   1:  PR[91,2] = PR[90,2] + 18.690;
   1:  PR[91,3] = PR[90,3] + 110.566;
   1:L PR[91] R[100]mm/sec CNT100;
   1:  PR[91,1] = PR[90,1] + -21.590;
   1:  PR[91,2] = PR[90,2] + 15.011;
   1:  PR[91,3] = PR[90,3] + 110.605;
   1:L PR[91] R[100]mm/sec CNT100;
   1:  PR[91,1] = PR[90,1] + -26.072;
   1:  PR[91,2] = PR[90,2] + 11.127;
   1:  PR[91,3] = PR[90,3] + 110.640;
   1:L PR[91] R[100]mm/sec CNT100;
   1:  PR[91,1] = PR[90,1] + -28.046;
   1:  PR[91,2] = PR[90,2] + 8.636;
   1:  PR[91,3] = PR[90,3] + 110.670;
   1:L PR[91] R[100]mm/sec CNT100;
   1:  PR[91,1] = PR[90,1] + -29.203;
   1:  PR[91,2] = PR[90,2] + 7.162;
   1:  PR[91,3] = PR[90,3] + 110.686;
   1:L PR[91] R[100]mm/sec CNT100;
   1:  PR[91] = PR[90];
   1:  PR[91,1] = PR[90,1] + -28.899;
   1:  PR[91,2] = PR[90,2] + 3.219;
   1:  PR[91,3] = PR[90,3] + 111.995;
   1:L PR[91] R[100]mm/sec CNT100;
   1:  PR[91,1] = PR[90,1] + -29.295;
   1:  PR[91,2] = PR[90,2] + 0.620;
   1:  PR[91,3] = PR[90,3] + 110.717;
   1:L PR[91] R[100]mm/sec CNT100;
   1:  PR[91,1] = PR[90,1] + -29.499;
   1:  PR[91,2] = PR[90,2] + -0.729;
   1:  PR[91,3] = PR[90,3] + 110.731;
   1:L PR[91] R[100]mm/sec CNT100;
   1:  PR[91,1] = PR[90,1] + -28.898;
   1:  PR[91,2] = PR[90,2] + -4.678;
   1:  PR[91,3] = PR[90,3] + 110.738;
   1:L PR[91] R[100]mm/sec CNT100;
   1:  PR[91,1] = PR[90,1] + -27.056;
   1:  PR[91,2] = PR[90,2] + -8.680;
   1:  PR[91,3] = PR[90,3] + 110.758;
   1:L PR[91] R[100]mm/sec CNT100;
   1:  PR[91,1] = PR[90,1] + -23.900;
   1:  PR[91,2] = PR[90,2] + -12.680;
   1:  PR[91,3] = PR[90,3] + 110.780;
   1:L PR[91] R[100]mm/sec CNT100;
   1:  PR[91,1] = PR[90,1] + -21.408;
   1:  PR[91,2] = PR[90,2] + -14.850;
   1:  PR[91,3] = PR[90,3] + 110.806;
   1:L PR[91] R[100]mm/sec CNT100;
   1:  PR[91,1] = PR[90,1] + -19.393;
   1:  PR[91,2] = PR[90,2] + -16.589;
   1:  PR[91,3] = PR[90,3] + 110.823;
   1:L PR[91] R[100]mm/sec CNT100;
   1:  PR[91,1] = PR[90,1] + -13.560;
   1:  PR[91,2] = PR[90,2] + -20.296;
   1:  PR[91,3] = PR[90,3] + 110.836;
   1:L PR[91] R[100]mm/sec CNT100;
   1:  PR[91,1] = PR[90,1] + -6.447;
   1:  PR[91,2] = PR[90,2] + -23.694;
   1:  PR[91,3] = PR[90,3] + 110.871;
   1:L PR[91] R[100]mm/sec CNT100;
   1:  PR[91,1] = PR[90,1] + -0.885;
   1:  PR[91,2] = PR[90,2] + -25.699;
   1:  PR[91,3] = PR[90,3] + 110.911;
   1:L PR[91] R[100]mm/sec CNT100;
   1:  PR[91,1] = PR[90,1] + 0.617;
   1:  PR[91,2] = PR[90,2] + -26.345;
   1:  PR[91,3] = PR[90,3] + 110.941;
   1:L PR[91] R[100]mm/sec CNT100;
   1:  PR[91,1] = PR[90,1] + 2.242;
   1:  PR[91,2] = PR[90,2] + -26.979;
   1:  PR[91,3] = PR[90,3] + 110.950;
   1:L PR[91] R[100]mm/sec CNT100;
   1:  PR[91,1] = PR[90,1] + 5.927;
   1:  PR[91,2] = PR[90,2] + -28.163;
   1:  PR[91,3] = PR[90,3] + 110.959;
   1:L PR[91] R[100]mm/sec CNT100;
   1:  PR[91,1] = PR[90,1] + 10.541;
   1:  PR[91,2] = PR[90,2] + -29.357;
   1:  PR[91,3] = PR[90,3] + 110.978;
   1:L PR[91] R[100]mm/sec CNT100;
   1:  PR[91,1] = PR[90,1] + 13.547;
   1:  PR[91,2] = PR[90,2] + -30.335;
   1:  PR[91,3] = PR[90,3] + 111.002;
   1:L PR[91] R[100]mm/sec CNT100;
   1:  PR[91,1] = PR[90,1] + 22.631;
   1:  PR[91,2] = PR[90,2] + -32.054;
   1:  PR[91,3] = PR[90,3] + 111.018;
   1:L PR[91] R[100]mm/sec CNT100;
   1:  PR[91,1] = PR[90,1] + 31.896;
   1:  PR[91,2] = PR[90,2] + -32.675;
   1:  PR[91,3] = PR[90,3] + 111.065;
   1:L PR[91] R[100]mm/sec CNT100;
   1:  PR[91,1] = PR[90,1] + 35.449;
   1:  PR[91,2] = PR[90,2] + -32.699;
   1:  PR[91,3] = PR[90,3] + 111.112;
   1:L PR[91] R[100]mm/sec CNT100;
   1:  PR[91,1] = PR[90,1] + 37.094;
   1:  PR[91,2] = PR[90,2] + -32.535;
   1:  PR[91,3] = PR[90,3] + 111.130;
   1:L PR[91] R[100]mm/sec CNT100;
   1:  PR[91,1] = PR[90,1] + 42.048;
   1:  PR[91,2] = PR[90,2] + -31.700;
   1:  PR[91,3] = PR[90,3] + 111.139;
   1:L PR[91] R[100]mm/sec CNT100;
   1:  PR[91,1] = PR[90,1] + 42.311;
   1:  PR[91,2] = PR[90,2] + -31.628;
   1:  PR[91,3] = PR[90,3] + 111.164;
   1:L PR[91] R[100]mm/sec CNT100;
   1:  PR[91,1] = PR[90,1] + 43.722;
   1:  PR[91,2] = PR[90,2] + -31.123;
   1:  PR[91,3] = PR[90,3] + 111.166;
   1:L PR[91] R[100]mm/sec CNT100;
   1:  PR[91,1] = PR[90,1] + 48.274;
   1:  PR[91,2] = PR[90,2] + -29.546;
   1:  PR[91,3] = PR[90,3] + 111.173;
   1:L PR[91] R[100]mm/sec CNT100;
   1:  PR[91,1] = PR[90,1] + 53.963;
   1:  PR[91,2] = PR[90,2] + -26.403;
   1:  PR[91,3] = PR[90,3] + 111.198;
   1:L PR[91] R[100]mm/sec CNT100;
   1:  PR[91,1] = PR[90,1] + 56.746;
   1:  PR[91,2] = PR[90,2] + -24.164;
   1:  PR[91,3] = PR[90,3] + 111.231;
   1:L PR[91] R[100]mm/sec CNT100;
   1:  PR[91,1] = PR[90,1] + 58.567;
   1:  PR[91,2] = PR[90,2] + -22.765;
   1:  PR[91,3] = PR[90,3] + 111.249;
   1:L PR[91] R[100]mm/sec CNT100;
   1:  PR[91,1] = PR[90,1] + 59.454;
   1:  PR[91,2] = PR[90,2] + -21.955;
   1:  PR[91,3] = PR[90,3] + 111.261;
   1:L PR[91] R[100]mm/sec CNT100;
   1:  PR[91,1] = PR[90,1] + 61.281;
   1:  PR[91,2] = PR[90,2] + -19.912;
   1:  PR[91,3] = PR[90,3] + 111.267;
   1:L PR[91] R[100]mm/sec CNT100;
   1:  PR[91,1] = PR[90,1] + 63.248;
   1:  PR[91,2] = PR[90,2] + -17.593;
   1:  PR[91,3] = PR[90,3] + 111.281;
   1:L PR[91] R[100]mm/sec CNT100;
   1:  PR[91,1] = PR[90,1] + 65.653;
   1:  PR[91,2] = PR[90,2] + -13.713;
   1:  PR[91,3] = PR[90,3] + 111.296;
   1:L PR[91] R[100]mm/sec CNT100;
   1:  PR[91,1] = PR[90,1] + 67.493;
   1:  PR[91,2] = PR[90,2] + -9.389;
   1:  PR[91,3] = PR[90,3] + 111.319;
   1:L PR[91] R[100]mm/sec CNT100;
   1:  PR[91,1] = PR[90,1] + 68.495;
   1:  PR[91,2] = PR[90,2] + -5.359;
   1:  PR[91,3] = PR[90,3] + 111.343;
   1:L PR[91] R[100]mm/sec CNT100;
   1:  PR[91,1] = PR[90,1] + 68.842;
   1:  PR[91,2] = PR[90,2] + -1.092;
   1:  PR[91,3] = PR[90,3] + 111.364;
   1:L PR[91] R[100]mm/sec CNT100;
   1:  PR[91,1] = PR[90,1] + 68.902;
   1:  PR[91,2] = PR[90,2] + -0.670;
   1:  PR[91,3] = PR[90,3] + 111.386;
   1:L PR[91] R[100]mm/sec CNT100;
   1:  PR[91,1] = PR[90,1] + 68.564;
   1:  PR[91,2] = PR[90,2] + 3.453;
   1:  PR[91,3] = PR[90,3] + 111.388;
   1:L PR[91] R[100]mm/sec CNT100;
   1:  PR[91,1] = PR[90,1] + 68.509;
   1:  PR[91,2] = PR[90,2] + 3.843;
   1:  PR[91,3] = PR[90,3] + 111.409;
   1:L PR[91] R[100]mm/sec CNT100;
   1:  PR[91,1] = PR[90,1] + 67.493;
   1:  PR[91,2] = PR[90,2] + 7.930;
   1:  PR[91,3] = PR[90,3] + 111.411;
   1:L PR[91] R[100]mm/sec CNT100;
   1:  PR[91,1] = PR[90,1] + 65.654;
   1:  PR[91,2] = PR[90,2] + 12.253;
   1:  PR[91,3] = PR[90,3] + 111.432;
   1:L PR[91] R[100]mm/sec CNT100;
   1:  PR[91,1] = PR[90,1] + 63.250;
   1:  PR[91,2] = PR[90,2] + 16.132;
   1:  PR[91,3] = PR[90,3] + 111.456;
   1:L PR[91] R[100]mm/sec CNT100;
   1:  PR[91,1] = PR[90,1] + 61.281;
   1:  PR[91,2] = PR[90,2] + 18.453;
   1:  PR[91,3] = PR[90,3] + 111.479;
   1:L PR[91] R[100]mm/sec CNT100;
   1:  PR[91,1] = PR[90,1] + 59.452;
   1:  PR[91,2] = PR[90,2] + 20.498;
   1:  PR[91,3] = PR[90,3] + 111.495;
   1:L PR[91] R[100]mm/sec CNT100;
   1:  PR[91,1] = PR[90,1] + 58.565;
   1:  PR[91,2] = PR[90,2] + 21.308;
   1:  PR[91,3] = PR[90,3] + 111.509;
   1:L PR[91] R[100]mm/sec CNT100;
   1:  PR[91,1] = PR[90,1] + 56.747;
   1:  PR[91,2] = PR[90,2] + 22.706;
   1:  PR[91,3] = PR[90,3] + 111.515;
   1:L PR[91] R[100]mm/sec CNT100;
   1:  PR[91,1] = PR[90,1] + 53.961;
   1:  PR[91,2] = PR[90,2] + 24.947;
   1:  PR[91,3] = PR[90,3] + 111.526;
   1:L PR[91] R[100]mm/sec CNT100;
   1:  PR[91,1] = PR[90,1] + 48.276;
   1:  PR[91,2] = PR[90,2] + 28.086;
   1:  PR[91,3] = PR[90,3] + 111.544;
   1:L PR[91] R[100]mm/sec CNT100;
   1:  PR[91,1] = PR[90,1] + 43.722;
   1:  PR[91,2] = PR[90,2] + 29.664;
   1:  PR[91,3] = PR[90,3] + 111.577;
   1:L PR[91] R[100]mm/sec CNT100;
   1:  PR[91,1] = PR[90,1] + 42.315;
   1:  PR[91,2] = PR[90,2] + 30.169;
   1:  PR[91,3] = PR[90,3] + 111.602;
   1:L PR[91] R[100]mm/sec CNT100;
   1:  PR[91,1] = PR[90,1] + 42.054;
   1:  PR[91,2] = PR[90,2] + 30.240;
   1:  PR[91,3] = PR[90,3] + 111.609;
   1:L PR[91] R[100]mm/sec CNT100;
   1:  PR[91,1] = PR[90,1] + 37.093;
   1:  PR[91,2] = PR[90,2] + 31.077;
   1:  PR[91,3] = PR[90,3] + 111.611;
   1:L PR[91] R[100]mm/sec CNT100;
   1:  PR[91,1] = PR[90,1] + 35.447;
   1:  PR[91,2] = PR[90,2] + 31.240;
   1:  PR[91,3] = PR[90,3] + 111.636;
   1:L PR[91] R[100]mm/sec CNT100;
   1:  PR[91,1] = PR[90,1] + 31.881;
   1:  PR[91,2] = PR[90,2] + 31.216;
   1:  PR[91,3] = PR[90,3] + 111.645;
   1:L PR[91] R[100]mm/sec CNT100;
   1:  PR[91,1] = PR[90,1] + 22.655;
   1:  PR[91,2] = PR[90,2] + 30.598;
   1:  PR[91,3] = PR[90,3] + 111.663;
   1:L PR[91] R[100]mm/sec CNT100;
   1:  PR[91,1] = PR[90,1] + 13.553;
   1:  PR[91,2] = PR[90,2] + 28.878;
   1:  PR[91,3] = PR[90,3] + 111.710;
   1:L PR[91] R[100]mm/sec CNT100;
   1:  PR[91,1] = PR[90,1] + 10.541;
   1:  PR[91,2] = PR[90,2] + 27.899;
   1:  PR[91,3] = PR[90,3] + 111.757;
   1:L PR[91] R[100]mm/sec CNT100;
   1:  PR[91,1] = PR[90,1] + 5.928;
   1:  PR[91,2] = PR[90,2] + 26.705;
   1:  PR[91,3] = PR[90,3] + 111.773;
   1:L PR[91] R[100]mm/sec CNT100;
   1:  PR[91,1] = PR[90,1] + 2.242;
   1:  PR[91,2] = PR[90,2] + 25.520;
   1:  PR[91,3] = PR[90,3] + 111.797;
   1:L PR[91] R[100]mm/sec CNT100;
   1:  PR[91,1] = PR[90,1] + 0.617;
   1:  PR[91,2] = PR[90,2] + 24.886;
   1:  PR[91,3] = PR[90,3] + 111.817;
   1:L PR[91] R[100]mm/sec CNT100;
   1:  PR[91,1] = PR[90,1] + -0.885;
   1:  PR[91,2] = PR[90,2] + 24.240;
   1:  PR[91,3] = PR[90,3] + 111.826;
   1:L PR[91] R[100]mm/sec CNT100;
   1:  PR[91,1] = PR[90,1] + -6.447;
   1:  PR[91,2] = PR[90,2] + 22.236;
   1:  PR[91,3] = PR[90,3] + 111.834;
   1:L PR[91] R[100]mm/sec CNT100;
   1:  PR[91,1] = PR[90,1] + -13.560;
   1:  PR[91,2] = PR[90,2] + 18.838;
   1:  PR[91,3] = PR[90,3] + 111.864;
   1:L PR[91] R[100]mm/sec CNT100;
   1:  PR[91,1] = PR[90,1] + -19.393;
   1:  PR[91,2] = PR[90,2] + 15.130;
   1:  PR[91,3] = PR[90,3] + 111.904;
   1:L PR[91] R[100]mm/sec CNT100;
   1:  PR[91,1] = PR[90,1] + -21.408;
   1:  PR[91,2] = PR[90,2] + 13.392;
   1:  PR[91,3] = PR[90,3] + 111.939;
   1:L PR[91] R[100]mm/sec CNT100;
   1:  PR[91,1] = PR[90,1] + -23.900;
   1:  PR[91,2] = PR[90,2] + 11.222;
   1:  PR[91,3] = PR[90,3] + 111.952;
   1:L PR[91] R[100]mm/sec CNT100;
   1:  PR[91,1] = PR[90,1] + -27.057;
   1:  PR[91,2] = PR[90,2] + 7.221;
   1:  PR[91,3] = PR[90,3] + 111.969;
   1:L PR[91] R[100]mm/sec CNT100;
   1:  PR[91] = PR[90];
   1:  PR[91,1] = PR[90,1] + -26.764;
   1:  PR[91,2] = PR[90,2] + 3.250;
   1:  PR[91,3] = PR[90,3] + 113.295;
   1:L PR[91] R[100]mm/sec CNT100;
   1:  PR[91,1] = PR[90,1] + -27.119;
   1:  PR[91,2] = PR[90,2] + 0.925;
   1:  PR[91,3] = PR[90,3] + 112.018;
   1:L PR[91] R[100]mm/sec CNT100;
   1:  PR[91,1] = PR[90,1] + -27.369;
   1:  PR[91,2] = PR[90,2] + -0.729;
   1:  PR[91,3] = PR[90,3] + 112.030;
   1:L PR[91] R[100]mm/sec CNT100;
   1:  PR[91,1] = PR[90,1] + -26.763;
   1:  PR[91,2] = PR[90,2] + -4.710;
   1:  PR[91,3] = PR[90,3] + 112.038;
   1:L PR[91] R[100]mm/sec CNT100;
   1:  PR[91,1] = PR[90,1] + -24.908;
   1:  PR[91,2] = PR[90,2] + -8.742;
   1:  PR[91,3] = PR[90,3] + 112.059;
   1:L PR[91] R[100]mm/sec CNT100;
   1:  PR[91,1] = PR[90,1] + -21.730;
   1:  PR[91,2] = PR[90,2] + -12.772;
   1:  PR[91,3] = PR[90,3] + 112.082;
   1:L PR[91] R[100]mm/sec CNT100;
   1:  PR[91,1] = PR[90,1] + -18.889;
   1:  PR[91,2] = PR[90,2] + -15.247;
   1:  PR[91,3] = PR[90,3] + 112.108;
   1:L PR[91] R[100]mm/sec CNT100;
   1:  PR[91,1] = PR[90,1] + -17.193;
   1:  PR[91,2] = PR[90,2] + -16.710;
   1:  PR[91,3] = PR[90,3] + 112.127;
   1:L PR[91] R[100]mm/sec CNT100;
   1:  PR[91,1] = PR[90,1] + -11.322;
   1:  PR[91,2] = PR[90,2] + -20.444;
   1:  PR[91,3] = PR[90,3] + 112.139;
   1:L PR[91] R[100]mm/sec CNT100;
   1:  PR[91,1] = PR[90,1] + -4.162;
   1:  PR[91,2] = PR[90,2] + -23.867;
   1:  PR[91,3] = PR[90,3] + 112.174;
   1:L PR[91] R[100]mm/sec CNT100;
   1:  PR[91,1] = PR[90,1] + -1.534;
   1:  PR[91,2] = PR[90,2] + -24.815;
   1:  PR[91,3] = PR[90,3] + 112.215;
   1:L PR[91] R[100]mm/sec CNT100;
   1:  PR[91,1] = PR[90,1] + 1.504;
   1:  PR[91,2] = PR[90,2] + -26.121;
   1:  PR[91,3] = PR[90,3] + 112.229;
   1:L PR[91] R[100]mm/sec CNT100;
   1:  PR[91,1] = PR[90,1] + 4.908;
   1:  PR[91,2] = PR[90,2] + -27.449;
   1:  PR[91,3] = PR[90,3] + 112.246;
   1:L PR[91] R[100]mm/sec CNT100;
   1:  PR[91,1] = PR[90,1] + 6.995;
   1:  PR[91,2] = PR[90,2] + -28.120;
   1:  PR[91,3] = PR[90,3] + 112.265;
   1:L PR[91] R[100]mm/sec CNT100;
   1:  PR[91,1] = PR[90,1] + 9.670;
   1:  PR[91,2] = PR[90,2] + -28.812;
   1:  PR[91,3] = PR[90,3] + 112.276;
   1:L PR[91] R[100]mm/sec CNT100;
   1:  PR[91,1] = PR[90,1] + 15.006;
   1:  PR[91,2] = PR[90,2] + -30.547;
   1:  PR[91,3] = PR[90,3] + 112.290;
   1:L PR[91] R[100]mm/sec CNT100;
   1:  PR[91,1] = PR[90,1] + 23.781;
   1:  PR[91,2] = PR[90,2] + -32.216;
   1:  PR[91,3] = PR[90,3] + 112.319;
   1:L PR[91] R[100]mm/sec CNT100;
   1:  PR[91,1] = PR[90,1] + 24.941;
   1:  PR[91,2] = PR[90,2] + -32.331;
   1:  PR[91,3] = PR[90,3] + 112.365;
   1:L PR[91] R[100]mm/sec CNT100;
   1:  PR[91,1] = PR[90,1] + 31.610;
   1:  PR[91,2] = PR[90,2] + -32.779;
   1:  PR[91,3] = PR[90,3] + 112.371;
   1:L PR[91] R[100]mm/sec CNT100;
   1:  PR[91,1] = PR[90,1] + 36.265;
   1:  PR[91,2] = PR[90,2] + -32.811;
   1:  PR[91,3] = PR[90,3] + 112.405;
   1:L PR[91] R[100]mm/sec CNT100;
   1:  PR[91,1] = PR[90,1] + 36.806;
   1:  PR[91,2] = PR[90,2] + -32.757;
   1:  PR[91,3] = PR[90,3] + 112.429;
   1:L PR[91] R[100]mm/sec CNT100;
   1:  PR[91,1] = PR[90,1] + 42.786;
   1:  PR[91,2] = PR[90,2] + -31.760;
   1:  PR[91,3] = PR[90,3] + 112.431;
   1:L PR[91] R[100]mm/sec CNT100;
   1:  PR[91,1] = PR[90,1] + 48.989;
   1:  PR[91,2] = PR[90,2] + -29.610;
   1:  PR[91,3] = PR[90,3] + 112.462;
   1:L PR[91] R[100]mm/sec CNT100;
   1:  PR[91,1] = PR[90,1] + 50.842;
   1:  PR[91,2] = PR[90,2] + -28.581;
   1:  PR[91,3] = PR[90,3] + 112.496;
   1:L PR[91] R[100]mm/sec CNT100;
   1:  PR[91,1] = PR[90,1] + 54.708;
   1:  PR[91,2] = PR[90,2] + -26.471;
   1:  PR[91,3] = PR[90,3] + 112.507;
   1:L PR[91] R[100]mm/sec CNT100;
   1:  PR[91,1] = PR[90,1] + 54.975;
   1:  PR[91,2] = PR[90,2] + -26.285;
   1:  PR[91,3] = PR[90,3] + 112.529;
   1:L PR[91] R[100]mm/sec CNT100;
   1:  PR[91,1] = PR[90,1] + 58.574;
   1:  PR[91,2] = PR[90,2] + -23.518;
   1:  PR[91,3] = PR[90,3] + 112.531;
   1:L PR[91] R[100]mm/sec CNT100;
   1:  PR[91,1] = PR[90,1] + 60.968;
   1:  PR[91,2] = PR[90,2] + -21.332;
   1:  PR[91,3] = PR[90,3] + 112.554;
   1:L PR[91] R[100]mm/sec CNT100;
   1:  PR[91,1] = PR[90,1] + 64.170;
   1:  PR[91,2] = PR[90,2] + -17.527;
   1:  PR[91,3] = PR[90,3] + 112.571;
   1:L PR[91] R[100]mm/sec CNT100;
   1:  PR[91,1] = PR[90,1] + 66.488;
   1:  PR[91,2] = PR[90,2] + -13.787;
   1:  PR[91,3] = PR[90,3] + 112.596;
   1:L PR[91] R[100]mm/sec CNT100;
   1:  PR[91,1] = PR[90,1] + 68.141;
   1:  PR[91,2] = PR[90,2] + -9.880;
   1:  PR[91,3] = PR[90,3] + 112.619;
   1:L PR[91] R[100]mm/sec CNT100;
   1:  PR[91,1] = PR[90,1] + 68.387;
   1:  PR[91,2] = PR[90,2] + -9.331;
   1:  PR[91,3] = PR[90,3] + 112.641;
   1:L PR[91] R[100]mm/sec CNT100;
   1:  PR[91,1] = PR[90,1] + 69.347;
   1:  PR[91,2] = PR[90,2] + -5.468;
   1:  PR[91,3] = PR[90,3] + 112.644;
   1:L PR[91] R[100]mm/sec CNT100;
   1:  PR[91,1] = PR[90,1] + 69.682;
   1:  PR[91,2] = PR[90,2] + -1.352;
   1:  PR[91,3] = PR[90,3] + 112.664;
   1:L PR[91] R[100]mm/sec CNT100;
   1:  PR[91,1] = PR[90,1] + 69.778;
   1:  PR[91,2] = PR[90,2] + -0.670;
   1:  PR[91,3] = PR[90,3] + 112.685;
   1:L PR[91] R[100]mm/sec CNT100;
   1:  PR[91,1] = PR[90,1] + 69.454;
   1:  PR[91,2] = PR[90,2] + 3.301;
   1:  PR[91,3] = PR[90,3] + 112.689;
   1:L PR[91] R[100]mm/sec CNT100;
   1:  PR[91,1] = PR[90,1] + 69.361;
   1:  PR[91,2] = PR[90,2] + 3.952;
   1:  PR[91,3] = PR[90,3] + 112.709;
   1:L PR[91] R[100]mm/sec CNT100;
   1:  PR[91,1] = PR[90,1] + 68.383;
   1:  PR[91,2] = PR[90,2] + 7.888;
   1:  PR[91,3] = PR[90,3] + 112.712;
   1:L PR[91] R[100]mm/sec CNT100;
   1:  PR[91,1] = PR[90,1] + 66.490;
   1:  PR[91,2] = PR[90,2] + 12.325;
   1:  PR[91,3] = PR[90,3] + 112.733;
   1:L PR[91] R[100]mm/sec CNT100;
   1:  PR[91,1] = PR[90,1] + 64.172;
   1:  PR[91,2] = PR[90,2] + 16.066;
   1:  PR[91,3] = PR[90,3] + 112.758;
   1:L PR[91] R[100]mm/sec CNT100;
   1:  PR[91,1] = PR[90,1] + 60.970;
   1:  PR[91,2] = PR[90,2] + 19.870;
   1:  PR[91,3] = PR[90,3] + 112.780;
   1:L PR[91] R[100]mm/sec CNT100;
   1:  PR[91,1] = PR[90,1] + 58.573;
   1:  PR[91,2] = PR[90,2] + 22.060;
   1:  PR[91,3] = PR[90,3] + 112.806;
   1:L PR[91] R[100]mm/sec CNT100;
   1:  PR[91,1] = PR[90,1] + 54.968;
   1:  PR[91,2] = PR[90,2] + 24.831;
   1:  PR[91,3] = PR[90,3] + 112.822;
   1:L PR[91] R[100]mm/sec CNT100;
   1:  PR[91,1] = PR[90,1] + 54.704;
   1:  PR[91,2] = PR[90,2] + 25.015;
   1:  PR[91,3] = PR[90,3] + 112.846;
   1:L PR[91] R[100]mm/sec CNT100;
   1:  PR[91,1] = PR[90,1] + 50.840;
   1:  PR[91,2] = PR[90,2] + 27.123;
   1:  PR[91,3] = PR[90,3] + 112.847;
   1:L PR[91] R[100]mm/sec CNT100;
   1:  PR[91,1] = PR[90,1] + 48.987;
   1:  PR[91,2] = PR[90,2] + 28.153;
   1:  PR[91,3] = PR[90,3] + 112.870;
   1:L PR[91] R[100]mm/sec CNT100;
   1:  PR[91,1] = PR[90,1] + 42.790;
   1:  PR[91,2] = PR[90,2] + 30.300;
   1:  PR[91,3] = PR[90,3] + 112.881;
   1:L PR[91] R[100]mm/sec CNT100;
   1:  PR[91,1] = PR[90,1] + 36.810;
   1:  PR[91,2] = PR[90,2] + 31.298;
   1:  PR[91,3] = PR[90,3] + 112.914;
   1:L PR[91] R[100]mm/sec CNT100;
   1:  PR[91,1] = PR[90,1] + 36.270;
   1:  PR[91,2] = PR[90,2] + 31.351;
   1:  PR[91,3] = PR[90,3] + 112.945;
   1:L PR[91] R[100]mm/sec CNT100;
   1:  PR[91,1] = PR[90,1] + 31.596;
   1:  PR[91,2] = PR[90,2] + 31.320;
   1:  PR[91,3] = PR[90,3] + 112.948;
   1:L PR[91] R[100]mm/sec CNT100;
   1:  PR[91,1] = PR[90,1] + 24.966;
   1:  PR[91,2] = PR[90,2] + 30.875;
   1:  PR[91,3] = PR[90,3] + 112.972;
   1:L PR[91] R[100]mm/sec CNT100;
   1:  PR[91,1] = PR[90,1] + 24.303;
   1:  PR[91,2] = PR[90,2] + 30.818;
   1:  PR[91,3] = PR[90,3] + 113.006;
   1:L PR[91] R[100]mm/sec CNT100;
   1:  PR[91,1] = PR[90,1] + 23.813;
   1:  PR[91,2] = PR[90,2] + 30.762;
   1:  PR[91,3] = PR[90,3] + 113.009;
   1:L PR[91] R[100]mm/sec CNT100;
   1:  PR[91,1] = PR[90,1] + 15.015;
   1:  PR[91,2] = PR[90,2] + 29.091;
   1:  PR[91,3] = PR[90,3] + 113.012;
   1:L PR[91] R[100]mm/sec CNT100;
   1:  PR[91,1] = PR[90,1] + 9.670;
   1:  PR[91,2] = PR[90,2] + 27.353;
   1:  PR[91,3] = PR[90,3] + 113.058;
   1:L PR[91] R[100]mm/sec CNT100;
   1:  PR[91,1] = PR[90,1] + 6.996;
   1:  PR[91,2] = PR[90,2] + 26.661;
   1:  PR[91,3] = PR[90,3] + 113.086;
   1:L PR[91] R[100]mm/sec CNT100;
   1:  PR[91,1] = PR[90,1] + 4.909;
   1:  PR[91,2] = PR[90,2] + 25.990;
   1:  PR[91,3] = PR[90,3] + 113.101;
   1:L PR[91] R[100]mm/sec CNT100;
   1:  PR[91,1] = PR[90,1] + 1.504;
   1:  PR[91,2] = PR[90,2] + 24.663;
   1:  PR[91,3] = PR[90,3] + 113.112;
   1:L PR[91] R[100]mm/sec CNT100;
   1:  PR[91,1] = PR[90,1] + -1.534;
   1:  PR[91,2] = PR[90,2] + 23.356;
   1:  PR[91,3] = PR[90,3] + 113.131;
   1:L PR[91] R[100]mm/sec CNT100;
   1:  PR[91,1] = PR[90,1] + -4.162;
   1:  PR[91,2] = PR[90,2] + 22.408;
   1:  PR[91,3] = PR[90,3] + 113.147;
   1:L PR[91] R[100]mm/sec CNT100;
   1:  PR[91,1] = PR[90,1] + -11.322;
   1:  PR[91,2] = PR[90,2] + 18.985;
   1:  PR[91,3] = PR[90,3] + 113.162;
   1:L PR[91] R[100]mm/sec CNT100;
   1:  PR[91,1] = PR[90,1] + -17.193;
   1:  PR[91,2] = PR[90,2] + 15.251;
   1:  PR[91,3] = PR[90,3] + 113.202;
   1:L PR[91] R[100]mm/sec CNT100;
   1:  PR[91,1] = PR[90,1] + -18.889;
   1:  PR[91,2] = PR[90,2] + 13.788;
   1:  PR[91,3] = PR[90,3] + 113.238;
   1:L PR[91] R[100]mm/sec CNT100;
   1:  PR[91,1] = PR[90,1] + -21.730;
   1:  PR[91,2] = PR[90,2] + 11.313;
   1:  PR[91,3] = PR[90,3] + 113.249;
   1:L PR[91] R[100]mm/sec CNT100;
   1:  PR[91,1] = PR[90,1] + -24.908;
   1:  PR[91,2] = PR[90,2] + 7.283;
   1:  PR[91,3] = PR[90,3] + 113.269;
   1:L PR[91] R[100]mm/sec CNT100;
   1:  PR[91] = PR[90];
   1:  PR[91,1] = PR[90,1] + -24.629;
   1:  PR[91,2] = PR[90,2] + 3.281;
   1:  PR[91,3] = PR[90,3] + 114.595;
   1:L PR[91] R[100]mm/sec CNT100;
   1:  PR[91,1] = PR[90,1] + -24.942;
   1:  PR[91,2] = PR[90,2] + 1.230;
   1:  PR[91,3] = PR[90,3] + 113.318;
   1:L PR[91] R[100]mm/sec CNT100;
   1:  PR[91,1] = PR[90,1] + -25.238;
   1:  PR[91,2] = PR[90,2] + -0.729;
   1:  PR[91,3] = PR[90,3] + 113.329;
   1:L PR[91] R[100]mm/sec CNT100;
   1:  PR[91,1] = PR[90,1] + -24.628;
   1:  PR[91,2] = PR[90,2] + -4.741;
   1:  PR[91,3] = PR[90,3] + 113.339;
   1:L PR[91] R[100]mm/sec CNT100;
   1:  PR[91,1] = PR[90,1] + -22.760;
   1:  PR[91,2] = PR[90,2] + -8.804;
   1:  PR[91,3] = PR[90,3] + 113.360;
   1:L PR[91] R[100]mm/sec CNT100;
   1:  PR[91,1] = PR[90,1] + -19.561;
   1:  PR[91,2] = PR[90,2] + -12.863;
   1:  PR[91,3] = PR[90,3] + 113.383;
   1:L PR[91] R[100]mm/sec CNT100;
   1:  PR[91,1] = PR[90,1] + -16.370;
   1:  PR[91,2] = PR[90,2] + -15.643;
   1:  PR[91,3] = PR[90,3] + 113.410;
   1:L PR[91] R[100]mm/sec CNT100;
   1:  PR[91,1] = PR[90,1] + -14.994;
   1:  PR[91,2] = PR[90,2] + -16.830;
   1:  PR[91,3] = PR[90,3] + 113.432;
   1:L PR[91] R[100]mm/sec CNT100;
   1:  PR[91,1] = PR[90,1] + -9.084;
   1:  PR[91,2] = PR[90,2] + -20.592;
   1:  PR[91,3] = PR[90,3] + 113.441;
   1:L PR[91] R[100]mm/sec CNT100;
   1:  PR[91,1] = PR[90,1] + -1.996;
   1:  PR[91,2] = PR[90,2] + -23.983;
   1:  PR[91,3] = PR[90,3] + 113.477;
   1:L PR[91] R[100]mm/sec CNT100;
   1:  PR[91,1] = PR[90,1] + -1.787;
   1:  PR[91,2] = PR[90,2] + -24.100;
   1:  PR[91,3] = PR[90,3] + 113.518;
   1:L PR[91] R[100]mm/sec CNT100;
   1:  PR[91,1] = PR[90,1] + 2.391;
   1:  PR[91,2] = PR[90,2] + -25.898;
   1:  PR[91,3] = PR[90,3] + 113.519;
   1:L PR[91] R[100]mm/sec CNT100;
   1:  PR[91,1] = PR[90,1] + 7.574;
   1:  PR[91,2] = PR[90,2] + -27.919;
   1:  PR[91,3] = PR[90,3] + 113.542;
   1:L PR[91] R[100]mm/sec CNT100;
   1:  PR[91,1] = PR[90,1] + 8.064;
   1:  PR[91,2] = PR[90,2] + -28.076;
   1:  PR[91,3] = PR[90,3] + 113.571;
   1:L PR[91] R[100]mm/sec CNT100;
   1:  PR[91,1] = PR[90,1] + 8.798;
   1:  PR[91,2] = PR[90,2] + -28.266;
   1:  PR[91,3] = PR[90,3] + 113.574;
   1:L PR[91] R[100]mm/sec CNT100;
   1:  PR[91,1] = PR[90,1] + 16.462;
   1:  PR[91,2] = PR[90,2] + -30.759;
   1:  PR[91,3] = PR[90,3] + 113.578;
   1:L PR[91] R[100]mm/sec CNT100;
   1:  PR[91,1] = PR[90,1] + 21.916;
   1:  PR[91,2] = PR[90,2] + -31.791;
   1:  PR[91,3] = PR[90,3] + 113.619;
   1:L PR[91] R[100]mm/sec CNT100;
   1:  PR[91,1] = PR[90,1] + 24.452;
   1:  PR[91,2] = PR[90,2] + -32.298;
   1:  PR[91,3] = PR[90,3] + 113.648;
   1:L PR[91] R[100]mm/sec CNT100;
   1:  PR[91,1] = PR[90,1] + 26.635;
   1:  PR[91,2] = PR[90,2] + -32.539;
   1:  PR[91,3] = PR[90,3] + 113.661;
   1:L PR[91] R[100]mm/sec CNT100;
   1:  PR[91,1] = PR[90,1] + 28.358;
   1:  PR[91,2] = PR[90,2] + -32.684;
   1:  PR[91,3] = PR[90,3] + 113.673;
   1:L PR[91] R[100]mm/sec CNT100;
   1:  PR[91,1] = PR[90,1] + 31.324;
   1:  PR[91,2] = PR[90,2] + -32.883;
   1:  PR[91,3] = PR[90,3] + 113.682;
   1:L PR[91] R[100]mm/sec CNT100;
   1:  PR[91,1] = PR[90,1] + 36.319;
   1:  PR[91,2] = PR[90,2] + -32.920;
   1:  PR[91,3] = PR[90,3] + 113.697;
   1:L PR[91] R[100]mm/sec CNT100;
   1:  PR[91,1] = PR[90,1] + 36.948;
   1:  PR[91,2] = PR[90,2] + -32.915;
   1:  PR[91,3] = PR[90,3] + 113.723;
   1:L PR[91] R[100]mm/sec CNT100;
   1:  PR[91,1] = PR[90,1] + 43.475;
   1:  PR[91,2] = PR[90,2] + -31.834;
   1:  PR[91,3] = PR[90,3] + 113.726;
   1:L PR[91] R[100]mm/sec CNT100;
   1:  PR[91,1] = PR[90,1] + 49.712;
   1:  PR[91,2] = PR[90,2] + -29.672;
   1:  PR[91,3] = PR[90,3] + 113.760;
   1:L PR[91] R[100]mm/sec CNT100;
   1:  PR[91,1] = PR[90,1] + 54.252;
   1:  PR[91,2] = PR[90,2] + -27.185;
   1:  PR[91,3] = PR[90,3] + 113.794;
   1:L PR[91] R[100]mm/sec CNT100;
   1:  PR[91,1] = PR[90,1] + 55.099;
   1:  PR[91,2] = PR[90,2] + -26.774;
   1:  PR[91,3] = PR[90,3] + 113.821;
   1:L PR[91] R[100]mm/sec CNT100;
   1:  PR[91,1] = PR[90,1] + 57.508;
   1:  PR[91,2] = PR[90,2] + -25.095;
   1:  PR[91,3] = PR[90,3] + 113.826;
   1:L PR[91] R[100]mm/sec CNT100;
   1:  PR[91,1] = PR[90,1] + 58.585;
   1:  PR[91,2] = PR[90,2] + -24.267;
   1:  PR[91,3] = PR[90,3] + 113.841;
   1:L PR[91] R[100]mm/sec CNT100;
   1:  PR[91,1] = PR[90,1] + 61.855;
   1:  PR[91,2] = PR[90,2] + -21.320;
   1:  PR[91,3] = PR[90,3] + 113.848;
   1:L PR[91] R[100]mm/sec CNT100;
   1:  PR[91,1] = PR[90,1] + 65.093;
   1:  PR[91,2] = PR[90,2] + -17.458;
   1:  PR[91,3] = PR[90,3] + 113.871;
   1:L PR[91] R[100]mm/sec CNT100;
   1:  PR[91,1] = PR[90,1] + 67.323;
   1:  PR[91,2] = PR[90,2] + -13.860;
   1:  PR[91,3] = PR[90,3] + 113.897;
   1:L PR[91] R[100]mm/sec CNT100;
   1:  PR[91,1] = PR[90,1] + 68.916;
   1:  PR[91,2] = PR[90,2] + -10.097;
   1:  PR[91,3] = PR[90,3] + 113.918;
   1:L PR[91] R[100]mm/sec CNT100;
   1:  PR[91,1] = PR[90,1] + 69.276;
   1:  PR[91,2] = PR[90,2] + -9.290;
   1:  PR[91,3] = PR[90,3] + 113.940;
   1:L PR[91] R[100]mm/sec CNT100;
   1:  PR[91,1] = PR[90,1] + 70.199;
   1:  PR[91,2] = PR[90,2] + -5.578;
   1:  PR[91,3] = PR[90,3] + 113.944;
   1:L PR[91] R[100]mm/sec CNT100;
   1:  PR[91,1] = PR[90,1] + 70.522;
   1:  PR[91,2] = PR[90,2] + -1.612;
   1:  PR[91,3] = PR[90,3] + 113.964;
   1:L PR[91] R[100]mm/sec CNT100;
   1:  PR[91,1] = PR[90,1] + 70.655;
   1:  PR[91,2] = PR[90,2] + -0.670;
   1:  PR[91,3] = PR[90,3] + 113.984;
   1:L PR[91] R[100]mm/sec CNT100;
   1:  PR[91,1] = PR[90,1] + 70.343;
   1:  PR[91,2] = PR[90,2] + 3.149;
   1:  PR[91,3] = PR[90,3] + 113.989;
   1:L PR[91] R[100]mm/sec CNT100;
   1:  PR[91,1] = PR[90,1] + 70.213;
   1:  PR[91,2] = PR[90,2] + 4.062;
   1:  PR[91,3] = PR[90,3] + 114.009;
   1:L PR[91] R[100]mm/sec CNT100;
   1:  PR[91,1] = PR[90,1] + 69.272;
   1:  PR[91,2] = PR[90,2] + 7.850;
   1:  PR[91,3] = PR[90,3] + 114.014;
   1:L PR[91] R[100]mm/sec CNT100;
   1:  PR[91,1] = PR[90,1] + 67.626;
   1:  PR[91,2] = PR[90,2] + 11.730;
   1:  PR[91,3] = PR[90,3] + 114.034;
   1:L PR[91] R[100]mm/sec CNT100;
   1:  PR[91,1] = PR[90,1] + 67.334;
   1:  PR[91,2] = PR[90,2] + 12.383;
   1:  PR[91,3] = PR[90,3] + 114.056;
   1:L PR[91] R[100]mm/sec CNT100;
   1:  PR[91,1] = PR[90,1] + 65.095;
   1:  PR[91,2] = PR[90,2] + 15.997;
   1:  PR[91,3] = PR[90,3] + 114.059;
   1:L PR[91] R[100]mm/sec CNT100;
   1:  PR[91,1] = PR[90,1] + 61.858;
   1:  PR[91,2] = PR[90,2] + 19.859;
   1:  PR[91,3] = PR[90,3] + 114.081;
   1:L PR[91] R[100]mm/sec CNT100;
   1:  PR[91,1] = PR[90,1] + 58.587;
   1:  PR[91,2] = PR[90,2] + 22.807;
   1:  PR[91,3] = PR[90,3] + 114.107;
   1:L PR[91] R[100]mm/sec CNT100;
   1:  PR[91,1] = PR[90,1] + 57.509;
   1:  PR[91,2] = PR[90,2] + 23.636;
   1:  PR[91,3] = PR[90,3] + 114.130;
   1:L PR[91] R[100]mm/sec CNT100;
   1:  PR[91,1] = PR[90,1] + 55.067;
   1:  PR[91,2] = PR[90,2] + 25.337;
   1:  PR[91,3] = PR[90,3] + 114.137;
   1:L PR[91] R[100]mm/sec CNT100;
   1:  PR[91,1] = PR[90,1] + 51.454;
   1:  PR[91,2] = PR[90,2] + 27.253;
   1:  PR[91,3] = PR[90,3] + 114.153;
   1:L PR[91] R[100]mm/sec CNT100;
   1:  PR[91,1] = PR[90,1] + 49.704;
   1:  PR[91,2] = PR[90,2] + 28.217;
   1:  PR[91,3] = PR[90,3] + 114.174;
   1:L PR[91] R[100]mm/sec CNT100;
   1:  PR[91,1] = PR[90,1] + 43.475;
   1:  PR[91,2] = PR[90,2] + 30.375;
   1:  PR[91,3] = PR[90,3] + 114.184;
   1:L PR[91] R[100]mm/sec CNT100;
   1:  PR[91,1] = PR[90,1] + 36.954;
   1:  PR[91,2] = PR[90,2] + 31.456;
   1:  PR[91,3] = PR[90,3] + 114.218;
   1:L PR[91] R[100]mm/sec CNT100;
   1:  PR[91,1] = PR[90,1] + 36.297;
   1:  PR[91,2] = PR[90,2] + 31.460;
   1:  PR[91,3] = PR[90,3] + 114.252;
   1:L PR[91] R[100]mm/sec CNT100;
   1:  PR[91,1] = PR[90,1] + 31.313;
   1:  PR[91,2] = PR[90,2] + 31.424;
   1:  PR[91,3] = PR[90,3] + 114.255;
   1:L PR[91] R[100]mm/sec CNT100;
   1:  PR[91,1] = PR[90,1] + 28.387;
   1:  PR[91,2] = PR[90,2] + 31.228;
   1:  PR[91,3] = PR[90,3] + 114.281;
   1:L PR[91] R[100]mm/sec CNT100;
   1:  PR[91,1] = PR[90,1] + 26.210;
   1:  PR[91,2] = PR[90,2] + 31.040;
   1:  PR[91,3] = PR[90,3] + 114.296;
   1:L PR[91] R[100]mm/sec CNT100;
   1:  PR[91,1] = PR[90,1] + 24.471;
   1:  PR[91,2] = PR[90,2] + 30.841;
   1:  PR[91,3] = PR[90,3] + 114.308;
   1:L PR[91] R[100]mm/sec CNT100;
   1:  PR[91,1] = PR[90,1] + 21.916;
   1:  PR[91,2] = PR[90,2] + 30.332;
   1:  PR[91,3] = PR[90,3] + 114.317;
   1:L PR[91] R[100]mm/sec CNT100;
   1:  PR[91,1] = PR[90,1] + 16.475;
   1:  PR[91,2] = PR[90,2] + 29.304;
   1:  PR[91,3] = PR[90,3] + 114.330;
   1:L PR[91] R[100]mm/sec CNT100;
   1:  PR[91,1] = PR[90,1] + 8.798;
   1:  PR[91,2] = PR[90,2] + 26.807;
   1:  PR[91,3] = PR[90,3] + 114.359;
   1:L PR[91] R[100]mm/sec CNT100;
   1:  PR[91,1] = PR[90,1] + 8.064;
   1:  PR[91,2] = PR[90,2] + 26.617;
   1:  PR[91,3] = PR[90,3] + 114.400;
   1:L PR[91] R[100]mm/sec CNT100;
   1:  PR[91,1] = PR[90,1] + 7.575;
   1:  PR[91,2] = PR[90,2] + 26.460;
   1:  PR[91,3] = PR[90,3] + 114.404;
   1:L PR[91] R[100]mm/sec CNT100;
   1:  PR[91,1] = PR[90,1] + 2.390;
   1:  PR[91,2] = PR[90,2] + 24.439;
   1:  PR[91,3] = PR[90,3] + 114.407;
   1:L PR[91] R[100]mm/sec CNT100;
   1:  PR[91,1] = PR[90,1] + -1.787;
   1:  PR[91,2] = PR[90,2] + 22.642;
   1:  PR[91,3] = PR[90,3] + 114.436;
   1:L PR[91] R[100]mm/sec CNT100;
   1:  PR[91,1] = PR[90,1] + -1.996;
   1:  PR[91,2] = PR[90,2] + 22.524;
   1:  PR[91,3] = PR[90,3] + 114.459;
   1:L PR[91] R[100]mm/sec CNT100;
   1:  PR[91,1] = PR[90,1] + -9.084;
   1:  PR[91,2] = PR[90,2] + 19.133;
   1:  PR[91,3] = PR[90,3] + 114.460;
   1:L PR[91] R[100]mm/sec CNT100;
   1:  PR[91,1] = PR[90,1] + -14.994;
   1:  PR[91,2] = PR[90,2] + 15.371;
   1:  PR[91,3] = PR[90,3] + 114.501;
   1:L PR[91] R[100]mm/sec CNT100;
   1:  PR[91,1] = PR[90,1] + -16.370;
   1:  PR[91,2] = PR[90,2] + 14.184;
   1:  PR[91,3] = PR[90,3] + 114.537;
   1:L PR[91] R[100]mm/sec CNT100;
   1:  PR[91,1] = PR[90,1] + -19.561;
   1:  PR[91,2] = PR[90,2] + 11.405;
   1:  PR[91,3] = PR[90,3] + 114.546;
   1:L PR[91] R[100]mm/sec CNT100;
   1:  PR[91,1] = PR[90,1] + -22.760;
   1:  PR[91,2] = PR[90,2] + 7.345;
   1:  PR[91,3] = PR[90,3] + 114.568;
   1:L PR[91] R[100]mm/sec CNT100;
   1:  PR[91] = PR[90];
   1:  PR[91,1] = PR[90,1] + -22.494;
   1:  PR[91,2] = PR[90,2] + 3.312;
   1:  PR[91,3] = PR[90,3] + 115.895;
   1:L PR[91] R[100]mm/sec CNT100;
   1:  PR[91,1] = PR[90,1] + -22.765;
   1:  PR[91,2] = PR[90,2] + 1.535;
   1:  PR[91,3] = PR[90,3] + 114.618;
   1:L PR[91] R[100]mm/sec CNT100;
   1:  PR[91,1] = PR[90,1] + -23.108;
   1:  PR[91,2] = PR[90,2] + -0.729;
   1:  PR[91,3] = PR[90,3] + 114.628;
   1:L PR[91] R[100]mm/sec CNT100;
   1:  PR[91,1] = PR[90,1] + -22.494;
   1:  PR[91,2] = PR[90,2] + -4.772;
   1:  PR[91,3] = PR[90,3] + 114.640;
   1:L PR[91] R[100]mm/sec CNT100;
   1:  PR[91,1] = PR[90,1] + -20.612;
   1:  PR[91,2] = PR[90,2] + -8.866;
   1:  PR[91,3] = PR[90,3] + 114.661;
   1:L PR[91] R[100]mm/sec CNT100;
   1:  PR[91,1] = PR[90,1] + -17.392;
   1:  PR[91,2] = PR[90,2] + -12.955;
   1:  PR[91,3] = PR[90,3] + 114.684;
   1:L PR[91] R[100]mm/sec CNT100;
   1:  PR[91,1] = PR[90,1] + -13.851;
   1:  PR[91,2] = PR[90,2] + -16.039;
   1:  PR[91,3] = PR[90,3] + 114.712;
   1:L PR[91] R[100]mm/sec CNT100;
   1:  PR[91,1] = PR[90,1] + -12.794;
   1:  PR[91,2] = PR[90,2] + -16.950;
   1:  PR[91,3] = PR[90,3] + 114.736;
   1:L PR[91] R[100]mm/sec CNT100;
   1:  PR[91,1] = PR[90,1] + -6.846;
   1:  PR[91,2] = PR[90,2] + -20.739;
   1:  PR[91,3] = PR[90,3] + 114.743;
   1:L PR[91] R[100]mm/sec CNT100;
   1:  PR[91,1] = PR[90,1] + -2.644;
   1:  PR[91,2] = PR[90,2] + -22.750;
   1:  PR[91,3] = PR[90,3] + 114.780;
   1:L PR[91] R[100]mm/sec CNT100;
   1:  PR[91,1] = PR[90,1] + 0.246;
   1:  PR[91,2] = PR[90,2] + -24.370;
   1:  PR[91,3] = PR[90,3] + 114.804;
   1:L PR[91] R[100]mm/sec CNT100;
   1:  PR[91,1] = PR[90,1] + 3.277;
   1:  PR[91,2] = PR[90,2] + -25.674;
   1:  PR[91,3] = PR[90,3] + 114.821;
   1:L PR[91] R[100]mm/sec CNT100;
   1:  PR[91,1] = PR[90,1] + 8.168;
   1:  PR[91,2] = PR[90,2] + -27.581;
   1:  PR[91,3] = PR[90,3] + 114.839;
   1:L PR[91] R[100]mm/sec CNT100;
   1:  PR[91,1] = PR[90,1] + 9.532;
   1:  PR[91,2] = PR[90,2] + -28.245;
   1:  PR[91,3] = PR[90,3] + 114.866;
   1:L PR[91] R[100]mm/sec CNT100;
   1:  PR[91,1] = PR[90,1] + 17.919;
   1:  PR[91,2] = PR[90,2] + -30.971;
   1:  PR[91,3] = PR[90,3] + 114.874;
   1:L PR[91] R[100]mm/sec CNT100;
   1:  PR[91,1] = PR[90,1] + 20.778;
   1:  PR[91,2] = PR[90,2] + -31.512;
   1:  PR[91,3] = PR[90,3] + 114.920;
   1:L PR[91] R[100]mm/sec CNT100;
   1:  PR[91,1] = PR[90,1] + 25.106;
   1:  PR[91,2] = PR[90,2] + -32.377;
   1:  PR[91,3] = PR[90,3] + 114.935;
   1:L PR[91] R[100]mm/sec CNT100;
   1:  PR[91,1] = PR[90,1] + 28.106;
   1:  PR[91,2] = PR[90,2] + -32.720;
   1:  PR[91,3] = PR[90,3] + 114.958;
   1:L PR[91] R[100]mm/sec CNT100;
   1:  PR[91,1] = PR[90,1] + 31.231;
   1:  PR[91,2] = PR[90,2] + -32.991;
   1:  PR[91,3] = PR[90,3] + 114.974;
   1:L PR[91] R[100]mm/sec CNT100;
   1:  PR[91,1] = PR[90,1] + 35.510;
   1:  PR[91,2] = PR[90,2] + -33.023;
   1:  PR[91,3] = PR[90,3] + 114.990;
   1:L PR[91] R[100]mm/sec CNT100;
   1:  PR[91,1] = PR[90,1] + 37.610;
   1:  PR[91,2] = PR[90,2] + -33.001;
   1:  PR[91,3] = PR[90,3] + 115.012;
   1:L PR[91] R[100]mm/sec CNT100;
   1:  PR[91,1] = PR[90,1] + 41.288;
   1:  PR[91,2] = PR[90,2] + -32.398;
   1:  PR[91,3] = PR[90,3] + 115.023;
   1:L PR[91] R[100]mm/sec CNT100;
   1:  PR[91,1] = PR[90,1] + 44.160;
   1:  PR[91,2] = PR[90,2] + -31.910;
   1:  PR[91,3] = PR[90,3] + 115.043;
   1:L PR[91] R[100]mm/sec CNT100;
   1:  PR[91,1] = PR[90,1] + 50.466;
   1:  PR[91,2] = PR[90,2] + -29.725;
   1:  PR[91,3] = PR[90,3] + 115.058;
   1:L PR[91] R[100]mm/sec CNT100;
   1:  PR[91,1] = PR[90,1] + 53.807;
   1:  PR[91,2] = PR[90,2] + -27.903;
   1:  PR[91,3] = PR[90,3] + 115.092;
   1:L PR[91] R[100]mm/sec CNT100;
   1:  PR[91,1] = PR[90,1] + 55.452;
   1:  PR[91,2] = PR[90,2] + -27.103;
   1:  PR[91,3] = PR[90,3] + 115.112;
   1:L PR[91] R[100]mm/sec CNT100;
   1:  PR[91,1] = PR[90,1] + 59.146;
   1:  PR[91,2] = PR[90,2] + -24.541;
   1:  PR[91,3] = PR[90,3] + 115.122;
   1:L PR[91] R[100]mm/sec CNT100;
   1:  PR[91,1] = PR[90,1] + 62.684;
   1:  PR[91,2] = PR[90,2] + -21.367;
   1:  PR[91,3] = PR[90,3] + 115.145;
   1:L PR[91] R[100]mm/sec CNT100;
   1:  PR[91,1] = PR[90,1] + 66.017;
   1:  PR[91,2] = PR[90,2] + -17.388;
   1:  PR[91,3] = PR[90,3] + 115.170;
   1:L PR[91] R[100]mm/sec CNT100;
   1:  PR[91,1] = PR[90,1] + 68.159;
   1:  PR[91,2] = PR[90,2] + -13.932;
   1:  PR[91,3] = PR[90,3] + 115.197;
   1:L PR[91] R[100]mm/sec CNT100;
   1:  PR[91,1] = PR[90,1] + 69.690;
   1:  PR[91,2] = PR[90,2] + -10.313;
   1:  PR[91,3] = PR[90,3] + 115.218;
   1:L PR[91] R[100]mm/sec CNT100;
   1:  PR[91,1] = PR[90,1] + 70.166;
   1:  PR[91,2] = PR[90,2] + -9.249;
   1:  PR[91,3] = PR[90,3] + 115.239;
   1:L PR[91] R[100]mm/sec CNT100;
   1:  PR[91,1] = PR[90,1] + 71.051;
   1:  PR[91,2] = PR[90,2] + -5.687;
   1:  PR[91,3] = PR[90,3] + 115.245;
   1:L PR[91] R[100]mm/sec CNT100;
   1:  PR[91,1] = PR[90,1] + 71.362;
   1:  PR[91,2] = PR[90,2] + -1.872;
   1:  PR[91,3] = PR[90,3] + 115.264;
   1:L PR[91] R[100]mm/sec CNT100;
   1:  PR[91,1] = PR[90,1] + 71.532;
   1:  PR[91,2] = PR[90,2] + -0.670;
   1:  PR[91,3] = PR[90,3] + 115.284;
   1:L PR[91] R[100]mm/sec CNT100;
   1:  PR[91,1] = PR[90,1] + 71.232;
   1:  PR[91,2] = PR[90,2] + 2.997;
   1:  PR[91,3] = PR[90,3] + 115.290;
   1:L PR[91] R[100]mm/sec CNT100;
   1:  PR[91,1] = PR[90,1] + 71.066;
   1:  PR[91,2] = PR[90,2] + 4.171;
   1:  PR[91,3] = PR[90,3] + 115.309;
   1:L PR[91] R[100]mm/sec CNT100;
   1:  PR[91,1] = PR[90,1] + 70.161;
   1:  PR[91,2] = PR[90,2] + 7.809;
   1:  PR[91,3] = PR[90,3] + 115.315;
   1:L PR[91] R[100]mm/sec CNT100;
   1:  PR[91,1] = PR[90,1] + 68.579;
   1:  PR[91,2] = PR[90,2] + 11.539;
   1:  PR[91,3] = PR[90,3] + 115.335;
   1:L PR[91] R[100]mm/sec CNT100;
   1:  PR[91,1] = PR[90,1] + 68.170;
   1:  PR[91,2] = PR[90,2] + 12.455;
   1:  PR[91,3] = PR[90,3] + 115.356;
   1:L PR[91] R[100]mm/sec CNT100;
   1:  PR[91,1] = PR[90,1] + 66.019;
   1:  PR[91,2] = PR[90,2] + 15.927;
   1:  PR[91,3] = PR[90,3] + 115.361;
   1:L PR[91] R[100]mm/sec CNT100;
   1:  PR[91,1] = PR[90,1] + 62.686;
   1:  PR[91,2] = PR[90,2] + 19.907;
   1:  PR[91,3] = PR[90,3] + 115.382;
   1:L PR[91] R[100]mm/sec CNT100;
   1:  PR[91,1] = PR[90,1] + 59.148;
   1:  PR[91,2] = PR[90,2] + 23.080;
   1:  PR[91,3] = PR[90,3] + 115.409;
   1:L PR[91] R[100]mm/sec CNT100;
   1:  PR[91,1] = PR[90,1] + 55.422;
   1:  PR[91,2] = PR[90,2] + 25.665;
   1:  PR[91,3] = PR[90,3] + 115.434;
   1:L PR[91] R[100]mm/sec CNT100;
   1:  PR[91,1] = PR[90,1] + 51.801;
   1:  PR[91,2] = PR[90,2] + 27.585;
   1:  PR[91,3] = PR[90,3] + 115.458;
   1:L PR[91] R[100]mm/sec CNT100;
   1:  PR[91,1] = PR[90,1] + 50.484;
   1:  PR[91,2] = PR[90,2] + 28.261;
   1:  PR[91,3] = PR[90,3] + 115.479;
   1:L PR[91] R[100]mm/sec CNT100;
   1:  PR[91,1] = PR[90,1] + 44.159;
   1:  PR[91,2] = PR[90,2] + 30.451;
   1:  PR[91,3] = PR[90,3] + 115.487;
   1:L PR[91] R[100]mm/sec CNT100;
   1:  PR[91,1] = PR[90,1] + 37.610;
   1:  PR[91,2] = PR[90,2] + 31.542;
   1:  PR[91,3] = PR[90,3] + 115.522;
   1:L PR[91] R[100]mm/sec CNT100;
   1:  PR[91,1] = PR[90,1] + 35.516;
   1:  PR[91,2] = PR[90,2] + 31.564;
   1:  PR[91,3] = PR[90,3] + 115.556;
   1:L PR[91] R[100]mm/sec CNT100;
   1:  PR[91,1] = PR[90,1] + 31.229;
   1:  PR[91,2] = PR[90,2] + 31.532;
   1:  PR[91,3] = PR[90,3] + 115.567;
   1:L PR[91] R[100]mm/sec CNT100;
   1:  PR[91,1] = PR[90,1] + 28.118;
   1:  PR[91,2] = PR[90,2] + 31.263;
   1:  PR[91,3] = PR[90,3] + 115.590;
   1:L PR[91] R[100]mm/sec CNT100;
   1:  PR[91,1] = PR[90,1] + 25.120;
   1:  PR[91,2] = PR[90,2] + 30.920;
   1:  PR[91,3] = PR[90,3] + 115.606;
   1:L PR[91] R[100]mm/sec CNT100;
   1:  PR[91,1] = PR[90,1] + 20.777;
   1:  PR[91,2] = PR[90,2] + 30.053;
   1:  PR[91,3] = PR[90,3] + 115.621;
   1:L PR[91] R[100]mm/sec CNT100;
   1:  PR[91,1] = PR[90,1] + 17.936;
   1:  PR[91,2] = PR[90,2] + 29.517;
   1:  PR[91,3] = PR[90,3] + 115.645;
   1:L PR[91] R[100]mm/sec CNT100;
   1:  PR[91,1] = PR[90,1] + 9.535;
   1:  PR[91,2] = PR[90,2] + 26.787;
   1:  PR[91,3] = PR[90,3] + 115.660;
   1:L PR[91] R[100]mm/sec CNT100;
   1:  PR[91,1] = PR[90,1] + 8.168;
   1:  PR[91,2] = PR[90,2] + 26.122;
   1:  PR[91,3] = PR[90,3] + 115.706;
   1:L PR[91] R[100]mm/sec CNT100;
   1:  PR[91,1] = PR[90,1] + 3.277;
   1:  PR[91,2] = PR[90,2] + 24.215;
   1:  PR[91,3] = PR[90,3] + 115.713;
   1:L PR[91] R[100]mm/sec CNT100;
   1:  PR[91,1] = PR[90,1] + 0.247;
   1:  PR[91,2] = PR[90,2] + 22.911;
   1:  PR[91,3] = PR[90,3] + 115.741;
   1:L PR[91] R[100]mm/sec CNT100;
   1:  PR[91,1] = PR[90,1] + -2.644;
   1:  PR[91,2] = PR[90,2] + 21.291;
   1:  PR[91,3] = PR[90,3] + 115.758;
   1:L PR[91] R[100]mm/sec CNT100;
   1:  PR[91,1] = PR[90,1] + -6.846;
   1:  PR[91,2] = PR[90,2] + 19.280;
   1:  PR[91,3] = PR[90,3] + 115.775;
   1:L PR[91] R[100]mm/sec CNT100;
   1:  PR[91,1] = PR[90,1] + -12.794;
   1:  PR[91,2] = PR[90,2] + 15.492;
   1:  PR[91,3] = PR[90,3] + 115.799;
   1:L PR[91] R[100]mm/sec CNT100;
   1:  PR[91,1] = PR[90,1] + -13.851;
   1:  PR[91,2] = PR[90,2] + 14.580;
   1:  PR[91,3] = PR[90,3] + 115.836;
   1:L PR[91] R[100]mm/sec CNT100;
   1:  PR[91,1] = PR[90,1] + -17.392;
   1:  PR[91,2] = PR[90,2] + 11.496;
   1:  PR[91,3] = PR[90,3] + 115.843;
   1:L PR[91] R[100]mm/sec CNT100;
   1:  PR[91,1] = PR[90,1] + -20.612;
   1:  PR[91,2] = PR[90,2] + 7.407;
   1:  PR[91,3] = PR[90,3] + 115.868;
   1:L PR[91] R[100]mm/sec CNT100;
   1:  PR[91] = PR[90];
   1:  PR[91,1] = PR[90,1] + -20.359;
   1:  PR[91,2] = PR[90,2] + 3.343;
   1:  PR[91,3] = PR[90,3] + 117.195;
   1:L PR[91] R[100]mm/sec CNT100;
   1:  PR[91,1] = PR[90,1] + -20.588;
   1:  PR[91,2] = PR[90,2] + 1.840;
   1:  PR[91,3] = PR[90,3] + 115.919;
   1:L PR[91] R[100]mm/sec CNT100;
   1:  PR[91,1] = PR[90,1] + -20.977;
   1:  PR[91,2] = PR[90,2] + -0.729;
   1:  PR[91,3] = PR[90,3] + 115.927;
   1:L PR[91] R[100]mm/sec CNT100;
   1:  PR[91,1] = PR[90,1] + -20.359;
   1:  PR[91,2] = PR[90,2] + -4.803;
   1:  PR[91,3] = PR[90,3] + 115.940;
   1:L PR[91] R[100]mm/sec CNT100;
   1:  PR[91,1] = PR[90,1] + -18.464;
   1:  PR[91,2] = PR[90,2] + -8.928;
   1:  PR[91,3] = PR[90,3] + 115.962;
   1:L PR[91] R[100]mm/sec CNT100;
   1:  PR[91,1] = PR[90,1] + -15.222;
   1:  PR[91,2] = PR[90,2] + -13.046;
   1:  PR[91,3] = PR[90,3] + 115.986;
   1:L PR[91] R[100]mm/sec CNT100;
   1:  PR[91,1] = PR[90,1] + -11.332;
   1:  PR[91,2] = PR[90,2] + -16.435;
   1:  PR[91,3] = PR[90,3] + 116.013;
   1:L PR[91] R[100]mm/sec CNT100;
   1:  PR[91,1] = PR[90,1] + -10.595;
   1:  PR[91,2] = PR[90,2] + -17.071;
   1:  PR[91,3] = PR[90,3] + 116.041;
   1:L PR[91] R[100]mm/sec CNT100;
   1:  PR[91,1] = PR[90,1] + -4.608;
   1:  PR[91,2] = PR[90,2] + -20.887;
   1:  PR[91,3] = PR[90,3] + 116.046;
   1:L PR[91] R[100]mm/sec CNT100;
   1:  PR[91,1] = PR[90,1] + -3.292;
   1:  PR[91,2] = PR[90,2] + -21.516;
   1:  PR[91,3] = PR[90,3] + 116.083;
   1:L PR[91] R[100]mm/sec CNT100;
   1:  PR[91,1] = PR[90,1] + 2.279;
   1:  PR[91,2] = PR[90,2] + -24.639;
   1:  PR[91,3] = PR[90,3] + 116.091;
   1:L PR[91] R[100]mm/sec CNT100;
   1:  PR[91,1] = PR[90,1] + 4.164;
   1:  PR[91,2] = PR[90,2] + -25.450;
   1:  PR[91,3] = PR[90,3] + 116.124;
   1:L PR[91] R[100]mm/sec CNT100;
   1:  PR[91,1] = PR[90,1] + 7.297;
   1:  PR[91,2] = PR[90,2] + -26.671;
   1:  PR[91,3] = PR[90,3] + 116.135;
   1:L PR[91] R[100]mm/sec CNT100;
   1:  PR[91,1] = PR[90,1] + 10.932;
   1:  PR[91,2] = PR[90,2] + -28.442;
   1:  PR[91,3] = PR[90,3] + 116.153;
   1:L PR[91] R[100]mm/sec CNT100;
   1:  PR[91,1] = PR[90,1] + 19.385;
   1:  PR[91,2] = PR[90,2] + -31.186;
   1:  PR[91,3] = PR[90,3] + 116.174;
   1:L PR[91] R[100]mm/sec CNT100;
   1:  PR[91,1] = PR[90,1] + 25.755;
   1:  PR[91,2] = PR[90,2] + -32.455;
   1:  PR[91,3] = PR[90,3] + 116.220;
   1:L PR[91] R[100]mm/sec CNT100;
   1:  PR[91,1] = PR[90,1] + 30.023;
   1:  PR[91,2] = PR[90,2] + -32.944;
   1:  PR[91,3] = PR[90,3] + 116.255;
   1:L PR[91] R[100]mm/sec CNT100;
   1:  PR[91,1] = PR[90,1] + 31.903;
   1:  PR[91,2] = PR[90,2] + -33.113;
   1:  PR[91,3] = PR[90,3] + 116.277;
   1:L PR[91] R[100]mm/sec CNT100;
   1:  PR[91,1] = PR[90,1] + 34.497;
   1:  PR[91,2] = PR[90,2] + -33.126;
   1:  PR[91,3] = PR[90,3] + 116.287;
   1:L PR[91] R[100]mm/sec CNT100;
   1:  PR[91,1] = PR[90,1] + 38.271;
   1:  PR[91,2] = PR[90,2] + -33.087;
   1:  PR[91,3] = PR[90,3] + 116.301;
   1:L PR[91] R[100]mm/sec CNT100;
   1:  PR[91,1] = PR[90,1] + 44.856;
   1:  PR[91,2] = PR[90,2] + -31.983;
   1:  PR[91,3] = PR[90,3] + 116.320;
   1:L PR[91] R[100]mm/sec CNT100;
   1:  PR[91,1] = PR[90,1] + 49.952;
   1:  PR[91,2] = PR[90,2] + -30.246;
   1:  PR[91,3] = PR[90,3] + 116.355;
   1:L PR[91] R[100]mm/sec CNT100;
   1:  PR[91,1] = PR[90,1] + 51.244;
   1:  PR[91,2] = PR[90,2] + -29.775;
   1:  PR[91,3] = PR[90,3] + 116.384;
   1:L PR[91] R[100]mm/sec CNT100;
   1:  PR[91,1] = PR[90,1] + 53.360;
   1:  PR[91,2] = PR[90,2] + -28.621;
   1:  PR[91,3] = PR[90,3] + 116.391;
   1:L PR[91] R[100]mm/sec CNT100;
   1:  PR[91,1] = PR[90,1] + 55.806;
   1:  PR[91,2] = PR[90,2] + -27.432;
   1:  PR[91,3] = PR[90,3] + 116.404;
   1:L PR[91] R[100]mm/sec CNT100;
   1:  PR[91,1] = PR[90,1] + 60.119;
   1:  PR[91,2] = PR[90,2] + -24.458;
   1:  PR[91,3] = PR[90,3] + 116.418;
   1:L PR[91] R[100]mm/sec CNT100;
   1:  PR[91,1] = PR[90,1] + 63.511;
   1:  PR[91,2] = PR[90,2] + -21.416;
   1:  PR[91,3] = PR[90,3] + 116.445;
   1:L PR[91] R[100]mm/sec CNT100;
   1:  PR[91,1] = PR[90,1] + 66.941;
   1:  PR[91,2] = PR[90,2] + -17.318;
   1:  PR[91,3] = PR[90,3] + 116.469;
   1:L PR[91] R[100]mm/sec CNT100;
   1:  PR[91,1] = PR[90,1] + 68.995;
   1:  PR[91,2] = PR[90,2] + -14.005;
   1:  PR[91,3] = PR[90,3] + 116.497;
   1:L PR[91] R[100]mm/sec CNT100;
   1:  PR[91,1] = PR[90,1] + 70.465;
   1:  PR[91,2] = PR[90,2] + -10.530;
   1:  PR[91,3] = PR[90,3] + 116.518;
   1:L PR[91] R[100]mm/sec CNT100;
   1:  PR[91,1] = PR[90,1] + 71.055;
   1:  PR[91,2] = PR[90,2] + -9.209;
   1:  PR[91,3] = PR[90,3] + 116.538;
   1:L PR[91] R[100]mm/sec CNT100;
   1:  PR[91,1] = PR[90,1] + 71.904;
   1:  PR[91,2] = PR[90,2] + -5.797;
   1:  PR[91,3] = PR[90,3] + 116.545;
   1:L PR[91] R[100]mm/sec CNT100;
   1:  PR[91,1] = PR[90,1] + 72.202;
   1:  PR[91,2] = PR[90,2] + -2.132;
   1:  PR[91,3] = PR[90,3] + 116.564;
   1:L PR[91] R[100]mm/sec CNT100;
   1:  PR[91,1] = PR[90,1] + 72.409;
   1:  PR[91,2] = PR[90,2] + -0.670;
   1:  PR[91,3] = PR[90,3] + 116.583;
   1:L PR[91] R[100]mm/sec CNT100;
   1:  PR[91,1] = PR[90,1] + 72.122;
   1:  PR[91,2] = PR[90,2] + 2.845;
   1:  PR[91,3] = PR[90,3] + 116.591;
   1:L PR[91] R[100]mm/sec CNT100;
   1:  PR[91,1] = PR[90,1] + 71.918;
   1:  PR[91,2] = PR[90,2] + 4.280;
   1:  PR[91,3] = PR[90,3] + 116.609;
   1:L PR[91] R[100]mm/sec CNT100;
   1:  PR[91,1] = PR[90,1] + 71.050;
   1:  PR[91,2] = PR[90,2] + 7.769;
   1:  PR[91,3] = PR[90,3] + 116.617;
   1:L PR[91] R[100]mm/sec CNT100;
   1:  PR[91,1] = PR[90,1] + 69.532;
   1:  PR[91,2] = PR[90,2] + 11.349;
   1:  PR[91,3] = PR[90,3] + 116.636;
   1:L PR[91] R[100]mm/sec CNT100;
   1:  PR[91,1] = PR[90,1] + 69.005;
   1:  PR[91,2] = PR[90,2] + 12.528;
   1:  PR[91,3] = PR[90,3] + 116.656;
   1:L PR[91] R[100]mm/sec CNT100;
   1:  PR[91,1] = PR[90,1] + 66.943;
   1:  PR[91,2] = PR[90,2] + 15.857;
   1:  PR[91,3] = PR[90,3] + 116.663;
   1:L PR[91] R[100]mm/sec CNT100;
   1:  PR[91,1] = PR[90,1] + 63.513;
   1:  PR[91,2] = PR[90,2] + 19.956;
   1:  PR[91,3] = PR[90,3] + 116.684;
   1:L PR[91] R[100]mm/sec CNT100;
   1:  PR[91,1] = PR[90,1] + 60.122;
   1:  PR[91,2] = PR[90,2] + 22.998;
   1:  PR[91,3] = PR[90,3] + 116.712;
   1:L PR[91] R[100]mm/sec CNT100;
   1:  PR[91,1] = PR[90,1] + 55.789;
   1:  PR[91,2] = PR[90,2] + 25.985;
   1:  PR[91,3] = PR[90,3] + 116.736;
   1:L PR[91] R[100]mm/sec CNT100;
   1:  PR[91,1] = PR[90,1] + 51.264;
   1:  PR[91,2] = PR[90,2] + 28.309;
   1:  PR[91,3] = PR[90,3] + 116.763;
   1:L PR[91] R[100]mm/sec CNT100;
   1:  PR[91,1] = PR[90,1] + 49.948;
   1:  PR[91,2] = PR[90,2] + 28.789;
   1:  PR[91,3] = PR[90,3] + 116.790;
   1:L PR[91] R[100]mm/sec CNT100;
   1:  PR[91,1] = PR[90,1] + 44.848;
   1:  PR[91,2] = PR[90,2] + 30.526;
   1:  PR[91,3] = PR[90,3] + 116.797;
   1:L PR[91] R[100]mm/sec CNT100;
   1:  PR[91,1] = PR[90,1] + 38.269;
   1:  PR[91,2] = PR[90,2] + 31.628;
   1:  PR[91,3] = PR[90,3] + 116.825;
   1:L PR[91] R[100]mm/sec CNT100;
   1:  PR[91,1] = PR[90,1] + 34.502;
   1:  PR[91,2] = PR[90,2] + 31.667;
   1:  PR[91,3] = PR[90,3] + 116.861;
   1:L PR[91] R[100]mm/sec CNT100;
   1:  PR[91,1] = PR[90,1] + 31.901;
   1:  PR[91,2] = PR[90,2] + 31.654;
   1:  PR[91,3] = PR[90,3] + 116.880;
   1:L PR[91] R[100]mm/sec CNT100;
   1:  PR[91,1] = PR[90,1] + 30.029;
   1:  PR[91,2] = PR[90,2] + 31.486;
   1:  PR[91,3] = PR[90,3] + 116.894;
   1:L PR[91] R[100]mm/sec CNT100;
   1:  PR[91,1] = PR[90,1] + 25.768;
   1:  PR[91,2] = PR[90,2] + 30.998;
   1:  PR[91,3] = PR[90,3] + 116.904;
   1:L PR[91] R[100]mm/sec CNT100;
   1:  PR[91,1] = PR[90,1] + 19.406;
   1:  PR[91,2] = PR[90,2] + 29.733;
   1:  PR[91,3] = PR[90,3] + 116.926;
   1:L PR[91] R[100]mm/sec CNT100;
   1:  PR[91,1] = PR[90,1] + 10.938;
   1:  PR[91,2] = PR[90,2] + 26.985;
   1:  PR[91,3] = PR[90,3] + 116.960;
   1:L PR[91] R[100]mm/sec CNT100;
   1:  PR[91,1] = PR[90,1] + 7.296;
   1:  PR[91,2] = PR[90,2] + 25.212;
   1:  PR[91,3] = PR[90,3] + 117.007;
   1:L PR[91] R[100]mm/sec CNT100;
   1:  PR[91,1] = PR[90,1] + 4.164;
   1:  PR[91,2] = PR[90,2] + 23.991;
   1:  PR[91,3] = PR[90,3] + 117.028;
   1:L PR[91] R[100]mm/sec CNT100;
   1:  PR[91,1] = PR[90,1] + 2.279;
   1:  PR[91,2] = PR[90,2] + 23.180;
   1:  PR[91,3] = PR[90,3] + 117.046;
   1:L PR[91] R[100]mm/sec CNT100;
   1:  PR[91,1] = PR[90,1] + -3.292;
   1:  PR[91,2] = PR[90,2] + 20.058;
   1:  PR[91,3] = PR[90,3] + 117.057;
   1:L PR[91] R[100]mm/sec CNT100;
   1:  PR[91,1] = PR[90,1] + -4.608;
   1:  PR[91,2] = PR[90,2] + 19.428;
   1:  PR[91,3] = PR[90,3] + 117.090;
   1:L PR[91] R[100]mm/sec CNT100;
   1:  PR[91,1] = PR[90,1] + -10.595;
   1:  PR[91,2] = PR[90,2] + 15.612;
   1:  PR[91,3] = PR[90,3] + 117.098;
   1:L PR[91] R[100]mm/sec CNT100;
   1:  PR[91,1] = PR[90,1] + -11.332;
   1:  PR[91,2] = PR[90,2] + 14.976;
   1:  PR[91,3] = PR[90,3] + 117.135;
   1:L PR[91] R[100]mm/sec CNT100;
   1:  PR[91,1] = PR[90,1] + -15.222;
   1:  PR[91,2] = PR[90,2] + 11.588;
   1:  PR[91,3] = PR[90,3] + 117.140;
   1:L PR[91] R[100]mm/sec CNT100;
   1:  PR[91,1] = PR[90,1] + -18.464;
   1:  PR[91,2] = PR[90,2] + 7.469;
   1:  PR[91,3] = PR[90,3] + 117.167;
   1:L PR[91] R[100]mm/sec CNT100;
   1:  PR[91] = PR[90];
   1:  PR[91,1] = PR[90,1] + -18.224;
   1:  PR[91,2] = PR[90,2] + 3.375;
   1:  PR[91,3] = PR[90,3] + 118.495;
   1:L PR[91] R[100]mm/sec CNT100;
   1:  PR[91,1] = PR[90,1] + -18.412;
   1:  PR[91,2] = PR[90,2] + 2.145;
   1:  PR[91,3] = PR[90,3] + 117.219;
   1:L PR[91] R[100]mm/sec CNT100;
   1:  PR[91,1] = PR[90,1] + -18.847;
   1:  PR[91,2] = PR[90,2] + -0.729;
   1:  PR[91,3] = PR[90,3] + 117.226;
   1:L PR[91] R[100]mm/sec CNT100;
   1:  PR[91,1] = PR[90,1] + -18.224;
   1:  PR[91,2] = PR[90,2] + -4.834;
   1:  PR[91,3] = PR[90,3] + 117.241;
   1:L PR[91] R[100]mm/sec CNT100;
   1:  PR[91,1] = PR[90,1] + -16.316;
   1:  PR[91,2] = PR[90,2] + -8.990;
   1:  PR[91,3] = PR[90,3] + 117.263;
   1:L PR[91] R[100]mm/sec CNT100;
   1:  PR[91,1] = PR[90,1] + -13.053;
   1:  PR[91,2] = PR[90,2] + -13.138;
   1:  PR[91,3] = PR[90,3] + 117.287;
   1:L PR[91] R[100]mm/sec CNT100;
   1:  PR[91,1] = PR[90,1] + -8.815;
   1:  PR[91,2] = PR[90,2] + -16.830;
   1:  PR[91,3] = PR[90,3] + 117.315;
   1:L PR[91] R[100]mm/sec CNT100;
   1:  PR[91,1] = PR[90,1] + -8.396;
   1:  PR[91,2] = PR[90,2] + -17.191;
   1:  PR[91,3] = PR[90,3] + 117.345;
   1:L PR[91] R[100]mm/sec CNT100;
   1:  PR[91,1] = PR[90,1] + -3.717;
   1:  PR[91,2] = PR[90,2] + -20.175;
   1:  PR[91,3] = PR[90,3] + 117.348;
   1:L PR[91] R[100]mm/sec CNT100;
   1:  PR[91,1] = PR[90,1] + -2.560;
   1:  PR[91,2] = PR[90,2] + -21.056;
   1:  PR[91,3] = PR[90,3] + 117.377;
   1:L PR[91] R[100]mm/sec CNT100;
   1:  PR[91,1] = PR[90,1] + 4.312;
   1:  PR[91,2] = PR[90,2] + -24.908;
   1:  PR[91,3] = PR[90,3] + 117.385;
   1:L PR[91] R[100]mm/sec CNT100;
   1:  PR[91,1] = PR[90,1] + 5.051;
   1:  PR[91,2] = PR[90,2] + -25.226;
   1:  PR[91,3] = PR[90,3] + 117.427;
   1:L PR[91] R[100]mm/sec CNT100;
   1:  PR[91,1] = PR[90,1] + 6.425;
   1:  PR[91,2] = PR[90,2] + -25.762;
   1:  PR[91,3] = PR[90,3] + 117.431;
   1:L PR[91] R[100]mm/sec CNT100;
   1:  PR[91,1] = PR[90,1] + 12.332;
   1:  PR[91,2] = PR[90,2] + -28.638;
   1:  PR[91,3] = PR[90,3] + 117.439;
   1:L PR[91] R[100]mm/sec CNT100;
   1:  PR[91,1] = PR[90,1] + 18.762;
   1:  PR[91,2] = PR[90,2] + -30.726;
   1:  PR[91,3] = PR[90,3] + 117.474;
   1:L PR[91] R[100]mm/sec CNT100;
   1:  PR[91,1] = PR[90,1] + 20.237;
   1:  PR[91,2] = PR[90,2] + -31.250;
   1:  PR[91,3] = PR[90,3] + 117.509;
   1:L PR[91] R[100]mm/sec CNT100;
   1:  PR[91,1] = PR[90,1] + 21.310;
   1:  PR[91,2] = PR[90,2] + -31.515;
   1:  PR[91,3] = PR[90,3] + 117.518;
   1:L PR[91] R[100]mm/sec CNT100;
   1:  PR[91,1] = PR[90,1] + 26.406;
   1:  PR[91,2] = PR[90,2] + -32.533;
   1:  PR[91,3] = PR[90,3] + 117.524;
   1:L PR[91] R[100]mm/sec CNT100;
   1:  PR[91,1] = PR[90,1] + 31.943;
   1:  PR[91,2] = PR[90,2] + -33.168;
   1:  PR[91,3] = PR[90,3] + 117.551;
   1:L PR[91] R[100]mm/sec CNT100;
   1:  PR[91,1] = PR[90,1] + 32.576;
   1:  PR[91,2] = PR[90,2] + -33.228;
   1:  PR[91,3] = PR[90,3] + 117.581;
   1:L PR[91] R[100]mm/sec CNT100;
   1:  PR[91,1] = PR[90,1] + 33.483;
   1:  PR[91,2] = PR[90,2] + -33.229;
   1:  PR[91,3] = PR[90,3] + 117.584;
   1:L PR[91] R[100]mm/sec CNT100;
   1:  PR[91,1] = PR[90,1] + 38.935;
   1:  PR[91,2] = PR[90,2] + -33.172;
   1:  PR[91,3] = PR[90,3] + 117.589;
   1:L PR[91] R[100]mm/sec CNT100;
   1:  PR[91,1] = PR[90,1] + 45.292;
   1:  PR[91,2] = PR[90,2] + -32.107;
   1:  PR[91,3] = PR[90,3] + 117.618;
   1:L PR[91] R[100]mm/sec CNT100;
   1:  PR[91,1] = PR[90,1] + 45.841;
   1:  PR[91,2] = PR[90,2] + -31.974;
   1:  PR[91,3] = PR[90,3] + 117.652;
   1:L PR[91] R[100]mm/sec CNT100;
   1:  PR[91,1] = PR[90,1] + 49.753;
   1:  PR[91,2] = PR[90,2] + -30.649;
   1:  PR[91,3] = PR[90,3] + 117.655;
   1:L PR[91] R[100]mm/sec CNT100;
   1:  PR[91,1] = PR[90,1] + 52.037;
   1:  PR[91,2] = PR[90,2] + -29.817;
   1:  PR[91,3] = PR[90,3] + 117.677;
   1:L PR[91] R[100]mm/sec CNT100;
   1:  PR[91,1] = PR[90,1] + 52.913;
   1:  PR[91,2] = PR[90,2] + -29.339;
   1:  PR[91,3] = PR[90,3] + 117.690;
   1:L PR[91] R[100]mm/sec CNT100;
   1:  PR[91,1] = PR[90,1] + 54.092;
   1:  PR[91,2] = PR[90,2] + -28.766;
   1:  PR[91,3] = PR[90,3] + 117.695;
   1:L PR[91] R[100]mm/sec CNT100;
   1:  PR[91,1] = PR[90,1] + 56.582;
   1:  PR[91,2] = PR[90,2] + -27.493;
   1:  PR[91,3] = PR[90,3] + 117.702;
   1:L PR[91] R[100]mm/sec CNT100;
   1:  PR[91,1] = PR[90,1] + 60.365;
   1:  PR[91,2] = PR[90,2] + -24.895;
   1:  PR[91,3] = PR[90,3] + 117.717;
   1:L PR[91] R[100]mm/sec CNT100;
   1:  PR[91,1] = PR[90,1] + 61.080;
   1:  PR[91,2] = PR[90,2] + -24.387;
   1:  PR[91,3] = PR[90,3] + 117.741;
   1:L PR[91] R[100]mm/sec CNT100;
   1:  PR[91,1] = PR[90,1] + 64.338;
   1:  PR[91,2] = PR[90,2] + -21.465;
   1:  PR[91,3] = PR[90,3] + 117.745;
   1:L PR[91] R[100]mm/sec CNT100;
   1:  PR[91,1] = PR[90,1] + 67.865;
   1:  PR[91,2] = PR[90,2] + -17.248;
   1:  PR[91,3] = PR[90,3] + 117.769;
   1:L PR[91] R[100]mm/sec CNT100;
   1:  PR[91,1] = PR[90,1] + 69.830;
   1:  PR[91,2] = PR[90,2] + -14.077;
   1:  PR[91,3] = PR[90,3] + 117.798;
   1:L PR[91] R[100]mm/sec CNT100;
   1:  PR[91,1] = PR[90,1] + 71.240;
   1:  PR[91,2] = PR[90,2] + -10.747;
   1:  PR[91,3] = PR[90,3] + 117.818;
   1:L PR[91] R[100]mm/sec CNT100;
   1:  PR[91,1] = PR[90,1] + 71.945;
   1:  PR[91,2] = PR[90,2] + -9.168;
   1:  PR[91,3] = PR[90,3] + 117.837;
   1:L PR[91] R[100]mm/sec CNT100;
   1:  PR[91,1] = PR[90,1] + 72.756;
   1:  PR[91,2] = PR[90,2] + -5.906;
   1:  PR[91,3] = PR[90,3] + 117.846;
   1:L PR[91] R[100]mm/sec CNT100;
   1:  PR[91,1] = PR[90,1] + 73.042;
   1:  PR[91,2] = PR[90,2] + -2.393;
   1:  PR[91,3] = PR[90,3] + 117.864;
   1:L PR[91] R[100]mm/sec CNT100;
   1:  PR[91,1] = PR[90,1] + 73.286;
   1:  PR[91,2] = PR[90,2] + -0.670;
   1:  PR[91,3] = PR[90,3] + 117.882;
   1:L PR[91] R[100]mm/sec CNT100;
   1:  PR[91,1] = PR[90,1] + 73.011;
   1:  PR[91,2] = PR[90,2] + 2.693;
   1:  PR[91,3] = PR[90,3] + 117.892;
   1:L PR[91] R[100]mm/sec CNT100;
   1:  PR[91,1] = PR[90,1] + 72.770;
   1:  PR[91,2] = PR[90,2] + 4.390;
   1:  PR[91,3] = PR[90,3] + 117.909;
   1:L PR[91] R[100]mm/sec CNT100;
   1:  PR[91,1] = PR[90,1] + 71.940;
   1:  PR[91,2] = PR[90,2] + 7.728;
   1:  PR[91,3] = PR[90,3] + 117.918;
   1:L PR[91] R[100]mm/sec CNT100;
   1:  PR[91,1] = PR[90,1] + 70.485;
   1:  PR[91,2] = PR[90,2] + 11.158;
   1:  PR[91,3] = PR[90,3] + 117.937;
   1:L PR[91] R[100]mm/sec CNT100;
   1:  PR[91,1] = PR[90,1] + 69.841;
   1:  PR[91,2] = PR[90,2] + 12.601;
   1:  PR[91,3] = PR[90,3] + 117.956;
   1:L PR[91] R[100]mm/sec CNT100;
   1:  PR[91,1] = PR[90,1] + 67.866;
   1:  PR[91,2] = PR[90,2] + 15.787;
   1:  PR[91,3] = PR[90,3] + 117.965;
   1:L PR[91] R[100]mm/sec CNT100;
   1:  PR[91,1] = PR[90,1] + 64.340;
   1:  PR[91,2] = PR[90,2] + 20.004;
   1:  PR[91,3] = PR[90,3] + 117.985;
   1:L PR[91] R[100]mm/sec CNT100;
   1:  PR[91,1] = PR[90,1] + 61.092;
   1:  PR[91,2] = PR[90,2] + 22.918;
   1:  PR[91,3] = PR[90,3] + 118.014;
   1:L PR[91] R[100]mm/sec CNT100;
   1:  PR[91,1] = PR[90,1] + 56.581;
   1:  PR[91,2] = PR[90,2] + 26.034;
   1:  PR[91,3] = PR[90,3] + 118.037;
   1:L PR[91] R[100]mm/sec CNT100;
   1:  PR[91,1] = PR[90,1] + 52.061;
   1:  PR[91,2] = PR[90,2] + 28.350;
   1:  PR[91,3] = PR[90,3] + 118.066;
   1:L PR[91] R[100]mm/sec CNT100;
   1:  PR[91,1] = PR[90,1] + 49.751;
   1:  PR[91,2] = PR[90,2] + 29.192;
   1:  PR[91,3] = PR[90,3] + 118.093;
   1:L PR[91] R[100]mm/sec CNT100;
   1:  PR[91,1] = PR[90,1] + 45.832;
   1:  PR[91,2] = PR[90,2] + 30.517;
   1:  PR[91,3] = PR[90,3] + 118.106;
   1:L PR[91] R[100]mm/sec CNT100;
   1:  PR[91,1] = PR[90,1] + 45.285;
   1:  PR[91,2] = PR[90,2] + 30.650;
   1:  PR[91,3] = PR[90,3] + 118.128;
   1:L PR[91] R[100]mm/sec CNT100;
   1:  PR[91,1] = PR[90,1] + 38.929;
   1:  PR[91,2] = PR[90,2] + 31.714;
   1:  PR[91,3] = PR[90,3] + 118.131;
   1:L PR[91] R[100]mm/sec CNT100;
   1:  PR[91,1] = PR[90,1] + 33.489;
   1:  PR[91,2] = PR[90,2] + 31.770;
   1:  PR[91,3] = PR[90,3] + 118.165;
   1:L PR[91] R[100]mm/sec CNT100;
   1:  PR[91,1] = PR[90,1] + 32.575;
   1:  PR[91,2] = PR[90,2] + 31.768;
   1:  PR[91,3] = PR[90,3] + 118.194;
   1:L PR[91] R[100]mm/sec CNT100;
   1:  PR[91,1] = PR[90,1] + 31.940;
   1:  PR[91,2] = PR[90,2] + 31.709;
   1:  PR[91,3] = PR[90,3] + 118.198;
   1:L PR[91] R[100]mm/sec CNT100;
   1:  PR[91,1] = PR[90,1] + 26.418;
   1:  PR[91,2] = PR[90,2] + 31.076;
   1:  PR[91,3] = PR[90,3] + 118.202;
   1:L PR[91] R[100]mm/sec CNT100;
   1:  PR[91,1] = PR[90,1] + 21.334;
   1:  PR[91,2] = PR[90,2] + 30.062;
   1:  PR[91,3] = PR[90,3] + 118.231;
   1:L PR[91] R[100]mm/sec CNT100;
   1:  PR[91,1] = PR[90,1] + 20.251;
   1:  PR[91,2] = PR[90,2] + 29.794;
   1:  PR[91,3] = PR[90,3] + 118.259;
   1:L PR[91] R[100]mm/sec CNT100;
   1:  PR[91,1] = PR[90,1] + 18.761;
   1:  PR[91,2] = PR[90,2] + 29.266;
   1:  PR[91,3] = PR[90,3] + 118.265;
   1:L PR[91] R[100]mm/sec CNT100;
   1:  PR[91,1] = PR[90,1] + 12.341;
   1:  PR[91,2] = PR[90,2] + 27.183;
   1:  PR[91,3] = PR[90,3] + 118.273;
   1:L PR[91] R[100]mm/sec CNT100;
   1:  PR[91,1] = PR[90,1] + 6.425;
   1:  PR[91,2] = PR[90,2] + 24.303;
   1:  PR[91,3] = PR[90,3] + 118.309;
   1:L PR[91] R[100]mm/sec CNT100;
   1:  PR[91,1] = PR[90,1] + 5.051;
   1:  PR[91,2] = PR[90,2] + 23.767;
   1:  PR[91,3] = PR[90,3] + 118.344;
   1:L PR[91] R[100]mm/sec CNT100;
   1:  PR[91,1] = PR[90,1] + 4.313;
   1:  PR[91,2] = PR[90,2] + 23.450;
   1:  PR[91,3] = PR[90,3] + 118.351;
   1:L PR[91] R[100]mm/sec CNT100;
   1:  PR[91,1] = PR[90,1] + -2.560;
   1:  PR[91,2] = PR[90,2] + 19.597;
   1:  PR[91,3] = PR[90,3] + 118.356;
   1:L PR[91] R[100]mm/sec CNT100;
   1:  PR[91,1] = PR[90,1] + -3.717;
   1:  PR[91,2] = PR[90,2] + 18.716;
   1:  PR[91,3] = PR[90,3] + 118.397;
   1:L PR[91] R[100]mm/sec CNT100;
   1:  PR[91,1] = PR[90,1] + -8.392;
   1:  PR[91,2] = PR[90,2] + 15.735;
   1:  PR[91,3] = PR[90,3] + 118.405;
   1:L PR[91] R[100]mm/sec CNT100;
   1:  PR[91,1] = PR[90,1] + -13.053;
   1:  PR[91,2] = PR[90,2] + 11.679;
   1:  PR[91,3] = PR[90,3] + 118.434;
   1:L PR[91] R[100]mm/sec CNT100;
   1:  PR[91,1] = PR[90,1] + -16.316;
   1:  PR[91,2] = PR[90,2] + 7.531;
   1:  PR[91,3] = PR[90,3] + 118.467;
   1:L PR[91] R[100]mm/sec CNT100;
   1:  PR[91] = PR[90];
   1:  PR[91,1] = PR[90,1] + -16.089;
   1:  PR[91,2] = PR[90,2] + 3.406;
   1:  PR[91,3] = PR[90,3] + 119.795;
   1:L PR[91] R[100]mm/sec CNT100;
   1:  PR[91,1] = PR[90,1] + -16.235;
   1:  PR[91,2] = PR[90,2] + 2.450;
   1:  PR[91,3] = PR[90,3] + 118.520;
   1:L PR[91] R[100]mm/sec CNT100;
   1:  PR[91,1] = PR[90,1] + -16.716;
   1:  PR[91,2] = PR[90,2] + -0.729;
   1:  PR[91,3] = PR[90,3] + 118.525;
   1:L PR[91] R[100]mm/sec CNT100;
   1:  PR[91,1] = PR[90,1] + -16.089;
   1:  PR[91,2] = PR[90,2] + -4.865;
   1:  PR[91,3] = PR[90,3] + 118.542;
   1:L PR[91] R[100]mm/sec CNT100;
   1:  PR[91,1] = PR[90,1] + -14.168;
   1:  PR[91,2] = PR[90,2] + -9.052;
   1:  PR[91,3] = PR[90,3] + 118.564;
   1:L PR[91] R[100]mm/sec CNT100;
   1:  PR[91,1] = PR[90,1] + -10.884;
   1:  PR[91,2] = PR[90,2] + -13.229;
   1:  PR[91,3] = PR[90,3] + 118.589;
   1:L PR[91] R[100]mm/sec CNT100;
   1:  PR[91,1] = PR[90,1] + -6.294;
   1:  PR[91,2] = PR[90,2] + -17.227;
   1:  PR[91,3] = PR[90,3] + 118.617;
   1:L PR[91] R[100]mm/sec CNT100;
   1:  PR[91,1] = PR[90,1] + -6.196;
   1:  PR[91,2] = PR[90,2] + -17.311;
   1:  PR[91,3] = PR[90,3] + 118.650;
   1:L PR[91] R[100]mm/sec CNT100;
   1:  PR[91,1] = PR[90,1] + -4.365;
   1:  PR[91,2] = PR[90,2] + -18.479;
   1:L PR[91] R[100]mm/sec CNT100;
   1:  PR[91,1] = PR[90,1] + -0.924;
   1:  PR[91,2] = PR[90,2] + -21.100;
   1:  PR[91,3] = PR[90,3] + 118.662;
   1:L PR[91] R[100]mm/sec CNT100;
   1:  PR[91,1] = PR[90,1] + 5.812;
   1:  PR[91,2] = PR[90,2] + -24.878;
   1:  PR[91,3] = PR[90,3] + 118.685;
   1:L PR[91] R[100]mm/sec CNT100;
   1:  PR[91,1] = PR[90,1] + 6.305;
   1:  PR[91,2] = PR[90,2] + -25.220;
   1:  PR[91,3] = PR[90,3] + 118.726;
   1:L PR[91] R[100]mm/sec CNT100;
   1:  PR[91,1] = PR[90,1] + 13.732;
   1:  PR[91,2] = PR[90,2] + -28.835;
   1:  PR[91,3] = PR[90,3] + 118.730;
   1:L PR[91] R[100]mm/sec CNT100;
   1:  PR[91,1] = PR[90,1] + 17.623;
   1:  PR[91,2] = PR[90,2] + -30.098;
   1:  PR[91,3] = PR[90,3] + 118.774;
   1:L PR[91] R[100]mm/sec CNT100;
   1:  PR[91,1] = PR[90,1] + 20.904;
   1:  PR[91,2] = PR[90,2] + -31.263;
   1:  PR[91,3] = PR[90,3] + 118.795;
   1:L PR[91] R[100]mm/sec CNT100;
   1:  PR[91,1] = PR[90,1] + 23.395;
   1:  PR[91,2] = PR[90,2] + -31.880;
   1:  PR[91,3] = PR[90,3] + 118.814;
   1:L PR[91] R[100]mm/sec CNT100;
   1:  PR[91,1] = PR[90,1] + 27.056;
   1:  PR[91,2] = PR[90,2] + -32.611;
   1:  PR[91,3] = PR[90,3] + 118.828;
   1:L PR[91] R[100]mm/sec CNT100;
   1:  PR[91,1] = PR[90,1] + 33.259;
   1:  PR[91,2] = PR[90,2] + -33.323;
   1:  PR[91,3] = PR[90,3] + 118.848;
   1:L PR[91] R[100]mm/sec CNT100;
   1:  PR[91,1] = PR[90,1] + 39.599;
   1:  PR[91,2] = PR[90,2] + -33.258;
   1:  PR[91,3] = PR[90,3] + 118.881;
   1:L PR[91] R[100]mm/sec CNT100;
   1:  PR[91,1] = PR[90,1] + 45.386;
   1:  PR[91,2] = PR[90,2] + -32.293;
   1:  PR[91,3] = PR[90,3] + 118.915;
   1:L PR[91] R[100]mm/sec CNT100;
   1:  PR[91,1] = PR[90,1] + 47.160;
   1:  PR[91,2] = PR[90,2] + -31.863;
   1:  PR[91,3] = PR[90,3] + 118.946;
   1:L PR[91] R[100]mm/sec CNT100;
   1:  PR[91,1] = PR[90,1] + 49.552;
   1:  PR[91,2] = PR[90,2] + -31.053;
   1:  PR[91,3] = PR[90,3] + 118.956;
   1:L PR[91] R[100]mm/sec CNT100;
   1:  PR[91,1] = PR[90,1] + 52.902;
   1:  PR[91,2] = PR[90,2] + -29.827;
   1:  PR[91,3] = PR[90,3] + 118.969;
   1:L PR[91] R[100]mm/sec CNT100;
   1:  PR[91,1] = PR[90,1] + 57.392;
   1:  PR[91,2] = PR[90,2] + -27.530;
   1:  PR[91,3] = PR[90,3] + 118.989;
   1:L PR[91] R[100]mm/sec CNT100;
   1:  PR[91,1] = PR[90,1] + 61.013;
   1:  PR[91,2] = PR[90,2] + -25.044;
   1:  PR[91,3] = PR[90,3] + 119.015;
   1:L PR[91] R[100]mm/sec CNT100;
   1:  PR[91,1] = PR[90,1] + 62.051;
   1:  PR[91,2] = PR[90,2] + -24.306;
   1:  PR[91,3] = PR[90,3] + 119.039;
   1:L PR[91] R[100]mm/sec CNT100;
   1:  PR[91,1] = PR[90,1] + 65.165;
   1:  PR[91,2] = PR[90,2] + -21.514;
   1:  PR[91,3] = PR[90,3] + 119.046;
   1:L PR[91] R[100]mm/sec CNT100;
   1:  PR[91,1] = PR[90,1] + 68.789;
   1:  PR[91,2] = PR[90,2] + -17.178;
   1:  PR[91,3] = PR[90,3] + 119.068;
   1:L PR[91] R[100]mm/sec CNT100;
   1:  PR[91,1] = PR[90,1] + 70.666;
   1:  PR[91,2] = PR[90,2] + -14.149;
   1:  PR[91,3] = PR[90,3] + 119.098;
   1:L PR[91] R[100]mm/sec CNT100;
   1:  PR[91,1] = PR[90,1] + 72.014;
   1:  PR[91,2] = PR[90,2] + -10.963;
   1:  PR[91,3] = PR[90,3] + 119.117;
   1:L PR[91] R[100]mm/sec CNT100;
   1:  PR[91,1] = PR[90,1] + 72.834;
   1:  PR[91,2] = PR[90,2] + -9.128;
   1:  PR[91,3] = PR[90,3] + 119.136;
   1:L PR[91] R[100]mm/sec CNT100;
   1:  PR[91,1] = PR[90,1] + 73.608;
   1:  PR[91,2] = PR[90,2] + -6.015;
   1:  PR[91,3] = PR[90,3] + 119.146;
   1:L PR[91] R[100]mm/sec CNT100;
   1:  PR[91,1] = PR[90,1] + 73.881;
   1:  PR[91,2] = PR[90,2] + -2.653;
   1:  PR[91,3] = PR[90,3] + 119.164;
   1:L PR[91] R[100]mm/sec CNT100;
   1:  PR[91,1] = PR[90,1] + 74.163;
   1:  PR[91,2] = PR[90,2] + -0.670;
   1:  PR[91,3] = PR[90,3] + 119.182;
   1:L PR[91] R[100]mm/sec CNT100;
   1:  PR[91,1] = PR[90,1] + 73.900;
   1:  PR[91,2] = PR[90,2] + 2.541;
   1:  PR[91,3] = PR[90,3] + 119.192;
   1:L PR[91] R[100]mm/sec CNT100;
   1:  PR[91,1] = PR[90,1] + 73.622;
   1:  PR[91,2] = PR[90,2] + 4.499;
   1:  PR[91,3] = PR[90,3] + 119.209;
   1:L PR[91] R[100]mm/sec CNT100;
   1:  PR[91,1] = PR[90,1] + 72.829;
   1:  PR[91,2] = PR[90,2] + 7.688;
   1:  PR[91,3] = PR[90,3] + 119.220;
   1:L PR[91] R[100]mm/sec CNT100;
   1:  PR[91,1] = PR[90,1] + 71.438;
   1:  PR[91,2] = PR[90,2] + 10.968;
   1:  PR[91,3] = PR[90,3] + 119.238;
   1:L PR[91] R[100]mm/sec CNT100;
   1:  PR[91,1] = PR[90,1] + 70.677;
   1:  PR[91,2] = PR[90,2] + 12.673;
   1:  PR[91,3] = PR[90,3] + 119.257;
   1:L PR[91] R[100]mm/sec CNT100;
   1:  PR[91,1] = PR[90,1] + 68.790;
   1:  PR[91,2] = PR[90,2] + 15.717;
   1:  PR[91,3] = PR[90,3] + 119.267;
   1:L PR[91] R[100]mm/sec CNT100;
   1:  PR[91,1] = PR[90,1] + 65.166;
   1:  PR[91,2] = PR[90,2] + 20.053;
   1:  PR[91,3] = PR[90,3] + 119.286;
   1:L PR[91] R[100]mm/sec CNT100;
   1:  PR[91,1] = PR[90,1] + 62.062;
   1:  PR[91,2] = PR[90,2] + 22.838;
   1:  PR[91,3] = PR[90,3] + 119.316;
   1:L PR[91] R[100]mm/sec CNT100;
   1:  PR[91,1] = PR[90,1] + 57.391;
   1:  PR[91,2] = PR[90,2] + 26.072;
   1:  PR[91,3] = PR[90,3] + 119.338;
   1:L PR[91] R[100]mm/sec CNT100;
   1:  PR[91,1] = PR[90,1] + 52.904;
   1:  PR[91,2] = PR[90,2] + 28.367;
   1:  PR[91,3] = PR[90,3] + 119.368;
   1:L PR[91] R[100]mm/sec CNT100;
   1:  PR[91,1] = PR[90,1] + 49.551;
   1:  PR[91,2] = PR[90,2] + 29.595;
   1:  PR[91,3] = PR[90,3] + 119.395;
   1:L PR[91] R[100]mm/sec CNT100;
   1:  PR[91,1] = PR[90,1] + 47.155;
   1:  PR[91,2] = PR[90,2] + 30.406;
   1:  PR[91,3] = PR[90,3] + 119.414;
   1:L PR[91] R[100]mm/sec CNT100;
   1:  PR[91,1] = PR[90,1] + 45.381;
   1:  PR[91,2] = PR[90,2] + 30.835;
   1:  PR[91,3] = PR[90,3] + 119.428;
   1:L PR[91] R[100]mm/sec CNT100;
   1:  PR[91,1] = PR[90,1] + 39.590;
   1:  PR[91,2] = PR[90,2] + 31.800;
   1:  PR[91,3] = PR[90,3] + 119.438;
   1:L PR[91] R[100]mm/sec CNT100;
   1:  PR[91,1] = PR[90,1] + 33.258;
   1:  PR[91,2] = PR[90,2] + 31.864;
   1:  PR[91,3] = PR[90,3] + 119.469;
   1:L PR[91] R[100]mm/sec CNT100;
   1:  PR[91,1] = PR[90,1] + 27.067;
   1:  PR[91,2] = PR[90,2] + 31.154;
   1:  PR[91,3] = PR[90,3] + 119.503;
   1:L PR[91] R[100]mm/sec CNT100;
   1:  PR[91,1] = PR[90,1] + 23.416;
   1:  PR[91,2] = PR[90,2] + 30.426;
   1:  PR[91,3] = PR[90,3] + 119.536;
   1:L PR[91] R[100]mm/sec CNT100;
   1:  PR[91,1] = PR[90,1] + 20.916;
   1:  PR[91,2] = PR[90,2] + 29.808;
   1:  PR[91,3] = PR[90,3] + 119.556;
   1:L PR[91] R[100]mm/sec CNT100;
   1:  PR[91,1] = PR[90,1] + 17.622;
   1:  PR[91,2] = PR[90,2] + 28.639;
   1:  PR[91,3] = PR[90,3] + 119.570;
   1:L PR[91] R[100]mm/sec CNT100;
   1:  PR[91,1] = PR[90,1] + 13.744;
   1:  PR[91,2] = PR[90,2] + 27.381;
   1:  PR[91,3] = PR[90,3] + 119.588;
   1:L PR[91] R[100]mm/sec CNT100;
   1:  PR[91,1] = PR[90,1] + 6.305;
   1:  PR[91,2] = PR[90,2] + 23.761;
   1:  PR[91,3] = PR[90,3] + 119.610;
   1:L PR[91] R[100]mm/sec CNT100;
   1:  PR[91,1] = PR[90,1] + 5.812;
   1:  PR[91,2] = PR[90,2] + 23.419;
   1:  PR[91,3] = PR[90,3] + 119.654;
   1:L PR[91] R[100]mm/sec CNT100;
   1:  PR[91,1] = PR[90,1] + -0.924;
   1:  PR[91,2] = PR[90,2] + 19.641;
   1:  PR[91,3] = PR[90,3] + 119.658;
   1:L PR[91] R[100]mm/sec CNT100;
   1:  PR[91,1] = PR[90,1] + -4.365;
   1:  PR[91,2] = PR[90,2] + 17.020;
   1:  PR[91,3] = PR[90,3] + 119.699;
   1:L PR[91] R[100]mm/sec CNT100;
   1:  PR[91,1] = PR[90,1] + -6.193;
   1:  PR[91,2] = PR[90,2] + 15.855;
   1:  PR[91,3] = PR[90,3] + 119.722;
   1:L PR[91] R[100]mm/sec CNT100;
   1:  PR[91,1] = PR[90,1] + -10.884;
   1:  PR[91,2] = PR[90,2] + 11.770;
   1:  PR[91,3] = PR[90,3] + 119.733;
   1:L PR[91] R[100]mm/sec CNT100;
   1:  PR[91,1] = PR[90,1] + -14.168;
   1:  PR[91,2] = PR[90,2] + 7.593;
   1:  PR[91,3] = PR[90,3] + 119.767;
   1:L PR[91] R[100]mm/sec CNT100;
   1:  PR[91] = PR[90];
   1:  PR[91,1] = PR[90,1] + -13.954;
   1:  PR[91,2] = PR[90,2] + 3.438;
   1:  PR[91,3] = PR[90,3] + 121.095;
   1:L PR[91] R[100]mm/sec CNT100;
   1:  PR[91,1] = PR[90,1] + -14.586;
   1:  PR[91,2] = PR[90,2] + -0.729;
   1:  PR[91,3] = PR[90,3] + 119.820;
   1:L PR[91] R[100]mm/sec CNT100;
   1:  PR[91,1] = PR[90,1] + -13.954;
   1:  PR[91,2] = PR[90,2] + -4.896;
   1:  PR[91,3] = PR[90,3] + 119.843;
   1:L PR[91] R[100]mm/sec CNT100;
   1:  PR[91,1] = PR[90,1] + -12.020;
   1:  PR[91,2] = PR[90,2] + -9.114;
   1:  PR[91,3] = PR[90,3] + 119.865;
   1:L PR[91] R[100]mm/sec CNT100;
   1:  PR[91,1] = PR[90,1] + -8.915;
   1:  PR[91,2] = PR[90,2] + -13.068;
   1:  PR[91,3] = PR[90,3] + 119.890;
   1:L PR[91] R[100]mm/sec CNT100;
   1:  PR[91,1] = PR[90,1] + -8.718;
   1:  PR[91,2] = PR[90,2] + -13.318;
   1:  PR[91,3] = PR[90,3] + 119.917;
   1:L PR[91] R[100]mm/sec CNT100;
   1:  PR[91,1] = PR[90,1] + -4.774;
   1:  PR[91,2] = PR[90,2] + -16.753;
   1:  PR[91,3] = PR[90,3] + 119.919;
   1:L PR[91] R[100]mm/sec CNT100;
   1:  PR[91,1] = PR[90,1] + -4.113;
   1:  PR[91,2] = PR[90,2] + -17.448;
   1:  PR[91,3] = PR[90,3] + 119.947;
   1:L PR[91] R[100]mm/sec CNT100;
   1:  PR[91,1] = PR[90,1] + -3.331;
   1:  PR[91,2] = PR[90,2] + -18.065;
   1:  PR[91,3] = PR[90,3] + 119.952;
   1:L PR[91] R[100]mm/sec CNT100;
   1:  PR[91,1] = PR[90,1] + 0.711;
   1:  PR[91,2] = PR[90,2] + -21.144;
   1:  PR[91,3] = PR[90,3] + 119.958;
   1:L PR[91] R[100]mm/sec CNT100;
   1:  PR[91,1] = PR[90,1] + 4.940;
   1:  PR[91,2] = PR[90,2] + -23.516;
   1:  PR[91,3] = PR[90,3] + 119.985;
   1:L PR[91] R[100]mm/sec CNT100;
   1:  PR[91,1] = PR[90,1] + 7.649;
   1:  PR[91,2] = PR[90,2] + -25.396;
   1:  PR[91,3] = PR[90,3] + 120.011;
   1:L PR[91] R[100]mm/sec CNT100;
   1:  PR[91,1] = PR[90,1] + 15.132;
   1:  PR[91,2] = PR[90,2] + -29.032;
   1:  PR[91,3] = PR[90,3] + 120.029;
   1:L PR[91] R[100]mm/sec CNT100;
   1:  PR[91,1] = PR[90,1] + 16.484;
   1:  PR[91,2] = PR[90,2] + -29.471;
   1:  PR[91,3] = PR[90,3] + 120.074;
   1:L PR[91] R[100]mm/sec CNT100;
   1:  PR[91,1] = PR[90,1] + 21.570;
   1:  PR[91,2] = PR[90,2] + -31.277;
   1:  PR[91,3] = PR[90,3] + 120.081;
   1:L PR[91] R[100]mm/sec CNT100;
   1:  PR[91,1] = PR[90,1] + 25.481;
   1:  PR[91,2] = PR[90,2] + -32.245;
   1:  PR[91,3] = PR[90,3] + 120.110;
   1:L PR[91] R[100]mm/sec CNT100;
   1:  PR[91,1] = PR[90,1] + 27.706;
   1:  PR[91,2] = PR[90,2] + -32.690;
   1:  PR[91,3] = PR[90,3] + 120.132;
   1:L PR[91] R[100]mm/sec CNT100;
   1:  PR[91,1] = PR[90,1] + 33.936;
   1:  PR[91,2] = PR[90,2] + -33.406;
   1:  PR[91,3] = PR[90,3] + 120.144;
   1:L PR[91] R[100]mm/sec CNT100;
   1:  PR[91,1] = PR[90,1] + 40.170;
   1:  PR[91,2] = PR[90,2] + -33.330;
   1:  PR[91,3] = PR[90,3] + 120.178;
   1:L PR[91] R[100]mm/sec CNT100;
   1:  PR[91,1] = PR[90,1] + 40.872;
   1:  PR[91,2] = PR[90,2] + -33.246;
   1:  PR[91,3] = PR[90,3] + 120.212;
   1:L PR[91] R[100]mm/sec CNT100;
   1:  PR[91,1] = PR[90,1] + 45.480;
   1:  PR[91,2] = PR[90,2] + -32.479;
   1:  PR[91,3] = PR[90,3] + 120.215;
   1:L PR[91] R[100]mm/sec CNT100;
   1:  PR[91,1] = PR[90,1] + 48.479;
   1:  PR[91,2] = PR[90,2] + -31.752;
   1:  PR[91,3] = PR[90,3] + 120.241;
   1:L PR[91] R[100]mm/sec CNT100;
   1:  PR[91,1] = PR[90,1] + 49.353;
   1:  PR[91,2] = PR[90,2] + -31.457;
   1:  PR[91,3] = PR[90,3] + 120.257;
   1:L PR[91] R[100]mm/sec CNT100;
   1:  PR[91,1] = PR[90,1] + 50.439;
   1:  PR[91,2] = PR[90,2] + -31.061;
   1:  PR[91,3] = PR[90,3] + 120.262;
   1:L PR[91] R[100]mm/sec CNT100;
   1:  PR[91,1] = PR[90,1] + 53.912;
   1:  PR[91,2] = PR[90,2] + -29.762;
   1:  PR[91,3] = PR[90,3] + 120.268;
   1:L PR[91] R[100]mm/sec CNT100;
   1:  PR[91,1] = PR[90,1] + 58.203;
   1:  PR[91,2] = PR[90,2] + -27.568;
   1:  PR[91,3] = PR[90,3] + 120.288;
   1:L PR[91] R[100]mm/sec CNT100;
   1:  PR[91,1] = PR[90,1] + 61.660;
   1:  PR[91,2] = PR[90,2] + -25.194;
   1:  PR[91,3] = PR[90,3] + 120.314;
   1:L PR[91] R[100]mm/sec CNT100;
   1:  PR[91,1] = PR[90,1] + 63.022;
   1:  PR[91,2] = PR[90,2] + -24.226;
   1:  PR[91,3] = PR[90,3] + 120.337;
   1:L PR[91] R[100]mm/sec CNT100;
   1:  PR[91,1] = PR[90,1] + 65.992;
   1:  PR[91,2] = PR[90,2] + -21.562;
   1:  PR[91,3] = PR[90,3] + 120.346;
   1:L PR[91] R[100]mm/sec CNT100;
   1:  PR[91,1] = PR[90,1] + 69.713;
   1:  PR[91,2] = PR[90,2] + -17.107;
   1:  PR[91,3] = PR[90,3] + 120.367;
   1:L PR[91] R[100]mm/sec CNT100;
   1:  PR[91,1] = PR[90,1] + 71.502;
   1:  PR[91,2] = PR[90,2] + -14.222;
   1:  PR[91,3] = PR[90,3] + 120.399;
   1:L PR[91] R[100]mm/sec CNT100;
   1:  PR[91,1] = PR[90,1] + 72.789;
   1:  PR[91,2] = PR[90,2] + -11.180;
   1:  PR[91,3] = PR[90,3] + 120.417;
   1:L PR[91] R[100]mm/sec CNT100;
   1:  PR[91,1] = PR[90,1] + 73.724;
   1:  PR[91,2] = PR[90,2] + -9.087;
   1:  PR[91,3] = PR[90,3] + 120.435;
   1:L PR[91] R[100]mm/sec CNT100;
   1:  PR[91,1] = PR[90,1] + 74.460;
   1:  PR[91,2] = PR[90,2] + -6.125;
   1:  PR[91,3] = PR[90,3] + 120.447;
   1:L PR[91] R[100]mm/sec CNT100;
   1:  PR[91,1] = PR[90,1] + 74.721;
   1:  PR[91,2] = PR[90,2] + -2.913;
   1:  PR[91,3] = PR[90,3] + 120.463;
   1:L PR[91] R[100]mm/sec CNT100;
   1:  PR[91,1] = PR[90,1] + 75.040;
   1:  PR[91,2] = PR[90,2] + -0.670;
   1:  PR[91,3] = PR[90,3] + 120.481;
   1:L PR[91] R[100]mm/sec CNT100;
   1:  PR[91,1] = PR[90,1] + 74.789;
   1:  PR[91,2] = PR[90,2] + 2.389;
   1:  PR[91,3] = PR[90,3] + 120.493;
   1:L PR[91] R[100]mm/sec CNT100;
   1:  PR[91,1] = PR[90,1] + 74.475;
   1:  PR[91,2] = PR[90,2] + 4.608;
   1:  PR[91,3] = PR[90,3] + 120.509;
   1:L PR[91] R[100]mm/sec CNT100;
   1:  PR[91,1] = PR[90,1] + 73.719;
   1:  PR[91,2] = PR[90,2] + 7.647;
   1:  PR[91,3] = PR[90,3] + 120.522;
   1:L PR[91] R[100]mm/sec CNT100;
   1:  PR[91,1] = PR[90,1] + 72.392;
   1:  PR[91,2] = PR[90,2] + 10.777;
   1:  PR[91,3] = PR[90,3] + 120.538;
   1:L PR[91] R[100]mm/sec CNT100;
   1:  PR[91,1] = PR[90,1] + 71.512;
   1:  PR[91,2] = PR[90,2] + 12.746;
   1:  PR[91,3] = PR[90,3] + 120.557;
   1:L PR[91] R[100]mm/sec CNT100;
   1:  PR[91,1] = PR[90,1] + 69.714;
   1:  PR[91,2] = PR[90,2] + 15.647;
   1:  PR[91,3] = PR[90,3] + 120.568;
   1:L PR[91] R[100]mm/sec CNT100;
   1:  PR[91,1] = PR[90,1] + 65.993;
   1:  PR[91,2] = PR[90,2] + 20.102;
   1:  PR[91,3] = PR[90,3] + 120.587;
   1:L PR[91] R[100]mm/sec CNT100;
   1:  PR[91,1] = PR[90,1] + 63.035;
   1:  PR[91,2] = PR[90,2] + 22.756;
   1:  PR[91,3] = PR[90,3] + 120.618;
   1:L PR[91] R[100]mm/sec CNT100;
   1:  PR[91,1] = PR[90,1] + 59.102;
   1:  PR[91,2] = PR[90,2] + 25.468;
   1:  PR[91,3] = PR[90,3] + 120.639;
   1:L PR[91] R[100]mm/sec CNT100;
   1:  PR[91,1] = PR[90,1] + 58.190;
   1:  PR[91,2] = PR[90,2] + 26.115;
   1:  PR[91,3] = PR[90,3] + 120.665;
   1:L PR[91] R[100]mm/sec CNT100;
   1:  PR[91,1] = PR[90,1] + 53.913;
   1:  PR[91,2] = PR[90,2] + 28.303;
   1:  PR[91,3] = PR[90,3] + 120.671;
   1:L PR[91] R[100]mm/sec CNT100;
   1:  PR[91,1] = PR[90,1] + 50.437;
   1:  PR[91,2] = PR[90,2] + 29.603;
   1:  PR[91,3] = PR[90,3] + 120.697;
   1:L PR[91] R[100]mm/sec CNT100;
   1:  PR[91,1] = PR[90,1] + 49.353;
   1:  PR[91,2] = PR[90,2] + 29.998;
   1:  PR[91,3] = PR[90,3] + 120.717;
   1:L PR[91] R[100]mm/sec CNT100;
   1:  PR[91,1] = PR[90,1] + 48.478;
   1:  PR[91,2] = PR[90,2] + 30.294;
   1:  PR[91,3] = PR[90,3] + 120.723;
   1:L PR[91] R[100]mm/sec CNT100;
   1:  PR[91,1] = PR[90,1] + 45.476;
   1:  PR[91,2] = PR[90,2] + 31.021;
   1:  PR[91,3] = PR[90,3] + 120.728;
   1:L PR[91] R[100]mm/sec CNT100;
   1:  PR[91,1] = PR[90,1] + 40.860;
   1:  PR[91,2] = PR[90,2] + 31.788;
   1:  PR[91,3] = PR[90,3] + 120.745;
   1:L PR[91] R[100]mm/sec CNT100;
   1:  PR[91,1] = PR[90,1] + 40.161;
   1:  PR[91,2] = PR[90,2] + 31.872;
   1:  PR[91,3] = PR[90,3] + 120.770;
   1:L PR[91] R[100]mm/sec CNT100;
   1:  PR[91,1] = PR[90,1] + 33.935;
   1:  PR[91,2] = PR[90,2] + 31.947;
   1:  PR[91,3] = PR[90,3] + 120.774;
   1:L PR[91] R[100]mm/sec CNT100;
   1:  PR[91,1] = PR[90,1] + 27.716;
   1:  PR[91,2] = PR[90,2] + 31.233;
   1:  PR[91,3] = PR[90,3] + 120.807;
   1:L PR[91] R[100]mm/sec CNT100;
   1:  PR[91,1] = PR[90,1] + 25.499;
   1:  PR[91,2] = PR[90,2] + 30.791;
   1:  PR[91,3] = PR[90,3] + 120.841;
   1:L PR[91] R[100]mm/sec CNT100;
   1:  PR[91,1] = PR[90,1] + 21.582;
   1:  PR[91,2] = PR[90,2] + 29.821;
   1:  PR[91,3] = PR[90,3] + 120.853;
   1:L PR[91] R[100]mm/sec CNT100;
   1:  PR[91,1] = PR[90,1] + 16.483;
   1:  PR[91,2] = PR[90,2] + 28.013;
   1:  PR[91,3] = PR[90,3] + 120.875;
   1:L PR[91] R[100]mm/sec CNT100;
   1:  PR[91,1] = PR[90,1] + 15.146;
   1:  PR[91,2] = PR[90,2] + 27.579;
   1:  PR[91,3] = PR[90,3] + 120.904;
   1:L PR[91] R[100]mm/sec CNT100;
   1:  PR[91,1] = PR[90,1] + 7.652;
   1:  PR[91,2] = PR[90,2] + 23.939;
   1:  PR[91,3] = PR[90,3] + 120.911;
   1:L PR[91] R[100]mm/sec CNT100;
   1:  PR[91,1] = PR[90,1] + 4.940;
   1:  PR[91,2] = PR[90,2] + 22.057;
   1:  PR[91,3] = PR[90,3] + 120.956;
   1:L PR[91] R[100]mm/sec CNT100;
   1:  PR[91,1] = PR[90,1] + 0.712;
   1:  PR[91,2] = PR[90,2] + 19.686;
   1:  PR[91,3] = PR[90,3] + 120.974;
   1:L PR[91] R[100]mm/sec CNT100;
   1:  PR[91,1] = PR[90,1] + -3.330;
   1:  PR[91,2] = PR[90,2] + 16.607;
   1:  PR[91,3] = PR[90,3] + 121.000;
   1:L PR[91] R[100]mm/sec CNT100;
   1:  PR[91,1] = PR[90,1] + -4.113;
   1:  PR[91,2] = PR[90,2] + 15.989;
   1:  PR[91,3] = PR[90,3] + 121.028;
   1:L PR[91] R[100]mm/sec CNT100;
   1:  PR[91,1] = PR[90,1] + -4.774;
   1:  PR[91,2] = PR[90,2] + 15.294;
   1:  PR[91,3] = PR[90,3] + 121.033;
   1:L PR[91] R[100]mm/sec CNT100;
   1:  PR[91,1] = PR[90,1] + -8.714;
   1:  PR[91,2] = PR[90,2] + 11.862;
   1:  PR[91,3] = PR[90,3] + 121.038;
   1:L PR[91] R[100]mm/sec CNT100;
   1:  PR[91,1] = PR[90,1] + -12.020;
   1:  PR[91,2] = PR[90,2] + 7.655;
   1:  PR[91,3] = PR[90,3] + 121.066;
   1:L PR[91] R[100]mm/sec CNT100;
   1:  PR[91] = PR[90];
   1:  PR[91,1] = PR[90,1] + -11.819;
   1:  PR[91,2] = PR[90,2] + 3.469;
   1:  PR[91,3] = PR[90,3] + 122.395;
   1:L PR[91] R[100]mm/sec CNT100;
   1:  PR[91,1] = PR[90,1] + -12.455;
   1:  PR[91,2] = PR[90,2] + -0.729;
   1:  PR[91,3] = PR[90,3] + 121.120;
   1:L PR[91] R[100]mm/sec CNT100;
   1:  PR[91,1] = PR[90,1] + -11.819;
   1:  PR[91,2] = PR[90,2] + -4.928;
   1:  PR[91,3] = PR[90,3] + 121.143;
   1:L PR[91] R[100]mm/sec CNT100;
   1:  PR[91,1] = PR[90,1] + -9.872;
   1:  PR[91,2] = PR[90,2] + -9.175;
   1:  PR[91,3] = PR[90,3] + 121.166;
   1:L PR[91] R[100]mm/sec CNT100;
   1:  PR[91,1] = PR[90,1] + -6.545;
   1:  PR[91,2] = PR[90,2] + -13.412;
   1:  PR[91,3] = PR[90,3] + 121.192;
   1:L PR[91] R[100]mm/sec CNT100;
   1:  PR[91,1] = PR[90,1] + -5.423;
   1:  PR[91,2] = PR[90,2] + -14.390;
   1:  PR[91,3] = PR[90,3] + 121.221;
   1:L PR[91] R[100]mm/sec CNT100;
   1:  PR[91,1] = PR[90,1] + -2.710;
   1:  PR[91,2] = PR[90,2] + -17.243;
   1:  PR[91,3] = PR[90,3] + 121.229;
   1:L PR[91] R[100]mm/sec CNT100;
   1:  PR[91,1] = PR[90,1] + 0.754;
   1:  PR[91,2] = PR[90,2] + -19.975;
   1:  PR[91,3] = PR[90,3] + 121.250;
   1:L PR[91] R[100]mm/sec CNT100;
   1:  PR[91,1] = PR[90,1] + 2.347;
   1:  PR[91,2] = PR[90,2] + -21.189;
   1:  PR[91,3] = PR[90,3] + 121.274;
   1:L PR[91] R[100]mm/sec CNT100;
   1:  PR[91,1] = PR[90,1] + 4.068;
   1:  PR[91,2] = PR[90,2] + -22.154;
   1:  PR[91,3] = PR[90,3] + 121.285;
   1:L PR[91] R[100]mm/sec CNT100;
   1:  PR[91,1] = PR[90,1] + 8.993;
   1:  PR[91,2] = PR[90,2] + -25.572;
   1:  PR[91,3] = PR[90,3] + 121.296;
   1:L PR[91] R[100]mm/sec CNT100;
   1:  PR[91,1] = PR[90,1] + 15.612;
   1:  PR[91,2] = PR[90,2] + -28.785;
   1:  PR[91,3] = PR[90,3] + 121.328;
   1:L PR[91] R[100]mm/sec CNT100;
   1:  PR[91,1] = PR[90,1] + 16.330;
   1:  PR[91,2] = PR[90,2] + -29.171;
   1:  PR[91,3] = PR[90,3] + 121.368;
   1:L PR[91] R[100]mm/sec CNT100;
   1:  PR[91,1] = PR[90,1] + 16.828;
   1:  PR[91,2] = PR[90,2] + -29.370;
   1:  PR[91,3] = PR[90,3] + 121.373;
   1:L PR[91] R[100]mm/sec CNT100;
   1:  PR[91,1] = PR[90,1] + 22.237;
   1:  PR[91,2] = PR[90,2] + -31.291;
   1:  PR[91,3] = PR[90,3] + 121.376;
   1:L PR[91] R[100]mm/sec CNT100;
   1:  PR[91,1] = PR[90,1] + 27.566;
   1:  PR[91,2] = PR[90,2] + -32.610;
   1:  PR[91,3] = PR[90,3] + 121.407;
   1:L PR[91] R[100]mm/sec CNT100;
   1:  PR[91,1] = PR[90,1] + 28.356;
   1:  PR[91,2] = PR[90,2] + -32.768;
   1:  PR[91,3] = PR[90,3] + 121.437;
   1:L PR[91] R[100]mm/sec CNT100;
   1:  PR[91,1] = PR[90,1] + 34.616;
   1:  PR[91,2] = PR[90,2] + -33.489;
   1:  PR[91,3] = PR[90,3] + 121.441;
   1:L PR[91] R[100]mm/sec CNT100;
   1:  PR[91,1] = PR[90,1] + 35.608;
   1:  PR[91,2] = PR[90,2] + -33.479;
   1:  PR[91,3] = PR[90,3] + 121.475;
   1:L PR[91] R[100]mm/sec CNT100;
   1:  PR[91,1] = PR[90,1] + 39.674;
   1:  PR[91,2] = PR[90,2] + -33.377;
   1:  PR[91,3] = PR[90,3] + 121.481;
   1:L PR[91] R[100]mm/sec CNT100;
   1:  PR[91,1] = PR[90,1] + 40.620;
   1:  PR[91,2] = PR[90,2] + -33.390;
   1:  PR[91,3] = PR[90,3] + 121.503;
   1:L PR[91] R[100]mm/sec CNT100;
   1:  PR[91,1] = PR[90,1] + 42.783;
   1:  PR[91,2] = PR[90,2] + -33.129;
   1:  PR[91,3] = PR[90,3] + 121.508;
   1:L PR[91] R[100]mm/sec CNT100;
   1:  PR[91,1] = PR[90,1] + 45.574;
   1:  PR[91,2] = PR[90,2] + -32.665;
   1:  PR[91,3] = PR[90,3] + 121.520;
   1:L PR[91] R[100]mm/sec CNT100;
   1:  PR[91,1] = PR[90,1] + 49.572;
   1:  PR[91,2] = PR[90,2] + -31.699;
   1:  PR[91,3] = PR[90,3] + 121.535;
   1:L PR[91] R[100]mm/sec CNT100;
   1:  PR[91,1] = PR[90,1] + 54.927;
   1:  PR[91,2] = PR[90,2] + -29.695;
   1:  PR[91,3] = PR[90,3] + 121.557;
   1:L PR[91] R[100]mm/sec CNT100;
   1:  PR[91,1] = PR[90,1] + 59.013;
   1:  PR[91,2] = PR[90,2] + -27.605;
   1:  PR[91,3] = PR[90,3] + 121.588;
   1:L PR[91] R[100]mm/sec CNT100;
   1:  PR[91,1] = PR[90,1] + 62.308;
   1:  PR[91,2] = PR[90,2] + -25.343;
   1:  PR[91,3] = PR[90,3] + 121.613;
   1:L PR[91] R[100]mm/sec CNT100;
   1:  PR[91,1] = PR[90,1] + 63.994;
   1:  PR[91,2] = PR[90,2] + -24.145;
   1:  PR[91,3] = PR[90,3] + 121.635;
   1:L PR[91] R[100]mm/sec CNT100;
   1:  PR[91,1] = PR[90,1] + 66.821;
   1:  PR[91,2] = PR[90,2] + -21.609;
   1:  PR[91,3] = PR[90,3] + 121.646;
   1:L PR[91] R[100]mm/sec CNT100;
   1:  PR[91,1] = PR[90,1] + 69.048;
   1:  PR[91,2] = PR[90,2] + -18.958;
   1:  PR[91,3] = PR[90,3] + 121.667;
   1:L PR[91] R[100]mm/sec CNT100;
   1:  PR[91,1] = PR[90,1] + 70.635;
   1:  PR[91,2] = PR[90,2] + -17.041;
   1:  PR[91,3] = PR[90,3] + 121.686;
   1:L PR[91] R[100]mm/sec CNT100;
   1:  PR[91,1] = PR[90,1] + 72.337;
   1:  PR[91,2] = PR[90,2] + -14.294;
   1:  PR[91,3] = PR[90,3] + 121.699;
   1:L PR[91] R[100]mm/sec CNT100;
   1:  PR[91,1] = PR[90,1] + 73.564;
   1:  PR[91,2] = PR[90,2] + -11.396;
   1:  PR[91,3] = PR[90,3] + 121.717;
   1:L PR[91] R[100]mm/sec CNT100;
   1:  PR[91,1] = PR[90,1] + 74.613;
   1:  PR[91,2] = PR[90,2] + -9.047;
   1:  PR[91,3] = PR[90,3] + 121.734;
   1:L PR[91] R[100]mm/sec CNT100;
   1:  PR[91,1] = PR[90,1] + 75.313;
   1:  PR[91,2] = PR[90,2] + -6.234;
   1:  PR[91,3] = PR[90,3] + 121.748;
   1:L PR[91] R[100]mm/sec CNT100;
   1:  PR[91,1] = PR[90,1] + 75.561;
   1:  PR[91,2] = PR[90,2] + -3.173;
   1:  PR[91,3] = PR[90,3] + 121.763;
   1:L PR[91] R[100]mm/sec CNT100;
   1:  PR[91,1] = PR[90,1] + 75.916;
   1:  PR[91,2] = PR[90,2] + -0.670;
   1:  PR[91,3] = PR[90,3] + 121.780;
   1:L PR[91] R[100]mm/sec CNT100;
   1:  PR[91,1] = PR[90,1] + 75.679;
   1:  PR[91,2] = PR[90,2] + 2.236;
   1:  PR[91,3] = PR[90,3] + 121.794;
   1:L PR[91] R[100]mm/sec CNT100;
   1:  PR[91,1] = PR[90,1] + 75.327;
   1:  PR[91,2] = PR[90,2] + 4.718;
   1:  PR[91,3] = PR[90,3] + 121.810;
   1:L PR[91] R[100]mm/sec CNT100;
   1:  PR[91,1] = PR[90,1] + 74.608;
   1:  PR[91,2] = PR[90,2] + 7.607;
   1:  PR[91,3] = PR[90,3] + 121.823;
   1:L PR[91] R[100]mm/sec CNT100;
   1:  PR[91,1] = PR[90,1] + 73.345;
   1:  PR[91,2] = PR[90,2] + 10.587;
   1:  PR[91,3] = PR[90,3] + 121.839;
   1:L PR[91] R[100]mm/sec CNT100;
   1:  PR[91,1] = PR[90,1] + 72.348;
   1:  PR[91,2] = PR[90,2] + 12.819;
   1:  PR[91,3] = PR[90,3] + 121.857;
   1:L PR[91] R[100]mm/sec CNT100;
   1:  PR[91,1] = PR[90,1] + 70.638;
   1:  PR[91,2] = PR[90,2] + 15.578;
   1:  PR[91,3] = PR[90,3] + 121.870;
   1:L PR[91] R[100]mm/sec CNT100;
   1:  PR[91,1] = PR[90,1] + 66.820;
   1:  PR[91,2] = PR[90,2] + 20.151;
   1:  PR[91,3] = PR[90,3] + 121.888;
   1:L PR[91] R[100]mm/sec CNT100;
   1:  PR[91,1] = PR[90,1] + 64.005;
   1:  PR[91,2] = PR[90,2] + 22.676;
   1:  PR[91,3] = PR[90,3] + 121.920;
   1:L PR[91] R[100]mm/sec CNT100;
   1:  PR[91,1] = PR[90,1] + 60.256;
   1:  PR[91,2] = PR[90,2] + 25.261;
   1:  PR[91,3] = PR[90,3] + 121.941;
   1:L PR[91] R[100]mm/sec CNT100;
   1:  PR[91,1] = PR[90,1] + 59.000;
   1:  PR[91,2] = PR[90,2] + 26.153;
   1:  PR[91,3] = PR[90,3] + 121.965;
   1:L PR[91] R[100]mm/sec CNT100;
   1:  PR[91,1] = PR[90,1] + 54.929;
   1:  PR[91,2] = PR[90,2] + 28.236;
   1:  PR[91,3] = PR[90,3] + 121.974;
   1:L PR[91] R[100]mm/sec CNT100;
   1:  PR[91,1] = PR[90,1] + 49.573;
   1:  PR[91,2] = PR[90,2] + 30.240;
   1:  PR[91,3] = PR[90,3] + 121.998;
   1:L PR[91] R[100]mm/sec CNT100;
   1:  PR[91,1] = PR[90,1] + 45.572;
   1:  PR[91,2] = PR[90,2] + 31.206;
   1:  PR[91,3] = PR[90,3] + 122.029;
   1:L PR[91] R[100]mm/sec CNT100;
   1:  PR[91,1] = PR[90,1] + 42.776;
   1:  PR[91,2] = PR[90,2] + 31.671;
   1:  PR[91,3] = PR[90,3] + 122.052;
   1:L PR[91] R[100]mm/sec CNT100;
   1:  PR[91,1] = PR[90,1] + 40.583;
   1:  PR[91,2] = PR[90,2] + 31.935;
   1:  PR[91,3] = PR[90,3] + 122.067;
   1:L PR[91] R[100]mm/sec CNT100;
   1:  PR[91,1] = PR[90,1] + 34.610;
   1:  PR[91,2] = PR[90,2] + 32.030;
   1:  PR[91,3] = PR[90,3] + 122.079;
   1:L PR[91] R[100]mm/sec CNT100;
   1:  PR[91,1] = PR[90,1] + 28.366;
   1:  PR[91,2] = PR[90,2] + 31.311;
   1:  PR[91,3] = PR[90,3] + 122.112;
   1:L PR[91] R[100]mm/sec CNT100;
   1:  PR[91,1] = PR[90,1] + 27.582;
   1:  PR[91,2] = PR[90,2] + 31.155;
   1:  PR[91,3] = PR[90,3] + 122.146;
   1:L PR[91] R[100]mm/sec CNT100;
   1:  PR[91,1] = PR[90,1] + 22.247;
   1:  PR[91,2] = PR[90,2] + 29.835;
   1:  PR[91,3] = PR[90,3] + 122.150;
   1:L PR[91] R[100]mm/sec CNT100;
   1:  PR[91,1] = PR[90,1] + 16.848;
   1:  PR[91,2] = PR[90,2] + 27.919;
   1:  PR[91,3] = PR[90,3] + 122.180;
   1:L PR[91] R[100]mm/sec CNT100;
   1:  PR[91,1] = PR[90,1] + 16.341;
   1:  PR[91,2] = PR[90,2] + 27.717;
   1:  PR[91,3] = PR[90,3] + 122.211;
   1:L PR[91] R[100]mm/sec CNT100;
   1:  PR[91,1] = PR[90,1] + 15.612;
   1:  PR[91,2] = PR[90,2] + 27.325;
   1:  PR[91,3] = PR[90,3] + 122.214;
   1:L PR[91] R[100]mm/sec CNT100;
   1:  PR[91,1] = PR[90,1] + 8.999;
   1:  PR[91,2] = PR[90,2] + 24.116;
   1:  PR[91,3] = PR[90,3] + 122.218;
   1:L PR[91] R[100]mm/sec CNT100;
   1:  PR[91,1] = PR[90,1] + 4.068;
   1:  PR[91,2] = PR[90,2] + 20.695;
   1:  PR[91,3] = PR[90,3] + 122.258;
   1:L PR[91] R[100]mm/sec CNT100;
   1:  PR[91,1] = PR[90,1] + 2.347;
   1:  PR[91,2] = PR[90,2] + 19.730;
   1:  PR[91,3] = PR[90,3] + 122.291;
   1:L PR[91] R[100]mm/sec CNT100;
   1:  PR[91,1] = PR[90,1] + 0.754;
   1:  PR[91,2] = PR[90,2] + 18.516;
   1:  PR[91,3] = PR[90,3] + 122.302;
   1:L PR[91] R[100]mm/sec CNT100;
   1:  PR[91,1] = PR[90,1] + -2.710;
   1:  PR[91,2] = PR[90,2] + 15.784;
   1:  PR[91,3] = PR[90,3] + 122.312;
   1:L PR[91] R[100]mm/sec CNT100;
   1:  PR[91,1] = PR[90,1] + -5.423;
   1:  PR[91,2] = PR[90,2] + 12.931;
   1:  PR[91,3] = PR[90,3] + 122.336;
   1:L PR[91] R[100]mm/sec CNT100;
   1:  PR[91,1] = PR[90,1] + -6.545;
   1:  PR[91,2] = PR[90,2] + 11.954;
   1:  PR[91,3] = PR[90,3] + 122.358;
   1:L PR[91] R[100]mm/sec CNT100;
   1:  PR[91,1] = PR[90,1] + -9.872;
   1:  PR[91,2] = PR[90,2] + 7.717;
   1:  PR[91,3] = PR[90,3] + 122.366;
   1:L PR[91] R[100]mm/sec CNT100;
   1:  PR[91] = PR[90];
   1:  PR[91,1] = PR[90,1] + -9.684;
   1:  PR[91,2] = PR[90,2] + 3.500;
   1:  PR[91,3] = PR[90,3] + 123.695;
   1:L PR[91] R[100]mm/sec CNT100;
   1:  PR[91,1] = PR[90,1] + -10.324;
   1:  PR[91,2] = PR[90,2] + -0.729;
   1:  PR[91,3] = PR[90,3] + 122.421;
   1:L PR[91] R[100]mm/sec CNT100;
   1:  PR[91,1] = PR[90,1] + -9.684;
   1:  PR[91,2] = PR[90,2] + -4.959;
   1:  PR[91,3] = PR[90,3] + 122.444;
   1:L PR[91] R[100]mm/sec CNT100;
   1:  PR[91,1] = PR[90,1] + -7.725;
   1:  PR[91,2] = PR[90,2] + -9.237;
   1:  PR[91,3] = PR[90,3] + 122.468;
   1:L PR[91] R[100]mm/sec CNT100;
   1:  PR[91,1] = PR[90,1] + -5.827;
   1:  PR[91,2] = PR[90,2] + -11.654;
   1:  PR[91,3] = PR[90,3] + 122.493;
   1:L PR[91] R[100]mm/sec CNT100;
   1:  PR[91,1] = PR[90,1] + -4.723;
   1:  PR[91,2] = PR[90,2] + -13.357;
   1:  PR[91,3] = PR[90,3] + 122.510;
   1:L PR[91] R[100]mm/sec CNT100;
   1:  PR[91,1] = PR[90,1] + -4.010;
   1:  PR[91,2] = PR[90,2] + -14.195;
   1:  PR[91,3] = PR[90,3] + 122.521;
   1:L PR[91] R[100]mm/sec CNT100;
   1:  PR[91,1] = PR[90,1] + -1.307;
   1:  PR[91,2] = PR[90,2] + -17.037;
   1:  PR[91,3] = PR[90,3] + 122.527;
   1:L PR[91] R[100]mm/sec CNT100;
   1:  PR[91,1] = PR[90,1] + 3.463;
   1:  PR[91,2] = PR[90,2] + -20.800;
   1:  PR[91,3] = PR[90,3] + 122.549;
   1:L PR[91] R[100]mm/sec CNT100;
   1:  PR[91,1] = PR[90,1] + 4.065;
   1:  PR[91,2] = PR[90,2] + -21.397;
   1:  PR[91,3] = PR[90,3] + 122.582;
   1:L PR[91] R[100]mm/sec CNT100;
   1:  PR[91,1] = PR[90,1] + 10.338;
   1:  PR[91,2] = PR[90,2] + -25.748;
   1:  PR[91,3] = PR[90,3] + 122.586;
   1:L PR[91] R[100]mm/sec CNT100;
   1:  PR[91,1] = PR[90,1] + 14.473;
   1:  PR[91,2] = PR[90,2] + -27.756;
   1:  PR[91,3] = PR[90,3] + 122.628;
   1:L PR[91] R[100]mm/sec CNT100;
   1:  PR[91,1] = PR[90,1] + 17.027;
   1:  PR[91,2] = PR[90,2] + -29.130;
   1:  PR[91,3] = PR[90,3] + 122.653;
   1:L PR[91] R[100]mm/sec CNT100;
   1:  PR[91,1] = PR[90,1] + 19.026;
   1:  PR[91,2] = PR[90,2] + -29.927;
   1:  PR[91,3] = PR[90,3] + 122.669;
   1:L PR[91] R[100]mm/sec CNT100;
   1:  PR[91,1] = PR[90,1] + 22.902;
   1:  PR[91,2] = PR[90,2] + -31.304;
   1:  PR[91,3] = PR[90,3] + 122.681;
   1:L PR[91] R[100]mm/sec CNT100;
   1:  PR[91,1] = PR[90,1] + 29.142;
   1:  PR[91,2] = PR[90,2] + -32.842;
   1:  PR[91,3] = PR[90,3] + 122.703;
   1:L PR[91] R[100]mm/sec CNT100;
   1:  PR[91,1] = PR[90,1] + 35.280;
   1:  PR[91,2] = PR[90,2] + -33.535;
   1:  PR[91,3] = PR[90,3] + 122.739;
   1:L PR[91] R[100]mm/sec CNT100;
   1:  PR[91,1] = PR[90,1] + 39.437;
   1:  PR[91,2] = PR[90,2] + -33.430;
   1:  PR[91,3] = PR[90,3] + 122.772;
   1:L PR[91] R[100]mm/sec CNT100;
   1:  PR[91,1] = PR[90,1] + 41.045;
   1:  PR[91,2] = PR[90,2] + -33.452;
   1:  PR[91,3] = PR[90,3] + 122.795;
   1:L PR[91] R[100]mm/sec CNT100;
   1:  PR[91,1] = PR[90,1] + 44.695;
   1:  PR[91,2] = PR[90,2] + -33.012;
   1:  PR[91,3] = PR[90,3] + 122.804;
   1:L PR[91] R[100]mm/sec CNT100;
   1:  PR[91,1] = PR[90,1] + 45.669;
   1:  PR[91,2] = PR[90,2] + -32.850;
   1:  PR[91,3] = PR[90,3] + 122.824;
   1:L PR[91] R[100]mm/sec CNT100;
   1:  PR[91,1] = PR[90,1] + 50.341;
   1:  PR[91,2] = PR[90,2] + -31.728;
   1:  PR[91,3] = PR[90,3] + 122.829;
   1:L PR[91] R[100]mm/sec CNT100;
   1:  PR[91,1] = PR[90,1] + 54.545;
   1:  PR[91,2] = PR[90,2] + -30.164;
   1:  PR[91,3] = PR[90,3] + 122.856;
   1:L PR[91] R[100]mm/sec CNT100;
   1:  PR[91,1] = PR[90,1] + 55.936;
   1:  PR[91,2] = PR[90,2] + -29.631;
   1:  PR[91,3] = PR[90,3] + 122.880;
   1:L PR[91] R[100]mm/sec CNT100;
   1:  PR[91,1] = PR[90,1] + 59.824;
   1:  PR[91,2] = PR[90,2] + -27.643;
   1:  PR[91,3] = PR[90,3] + 122.888;
   1:L PR[91] R[100]mm/sec CNT100;
   1:  PR[91,1] = PR[90,1] + 62.956;
   1:  PR[91,2] = PR[90,2] + -25.492;
   1:  PR[91,3] = PR[90,3] + 122.912;
   1:L PR[91] R[100]mm/sec CNT100;
   1:  PR[91,1] = PR[90,1] + 64.965;
   1:  PR[91,2] = PR[90,2] + -24.064;
   1:  PR[91,3] = PR[90,3] + 122.933;
   1:L PR[91] R[100]mm/sec CNT100;
   1:  PR[91,1] = PR[90,1] + 67.649;
   1:  PR[91,2] = PR[90,2] + -21.657;
   1:  PR[91,3] = PR[90,3] + 122.946;
   1:L PR[91] R[100]mm/sec CNT100;
   1:  PR[91,1] = PR[90,1] + 69.765;
   1:  PR[91,2] = PR[90,2] + -19.137;
   1:  PR[91,3] = PR[90,3] + 122.966;
   1:L PR[91] R[100]mm/sec CNT100;
   1:  PR[91,1] = PR[90,1] + 71.559;
   1:  PR[91,2] = PR[90,2] + -16.970;
   1:  PR[91,3] = PR[90,3] + 122.984;
   1:L PR[91] R[100]mm/sec CNT100;
   1:  PR[91,1] = PR[90,1] + 73.173;
   1:  PR[91,2] = PR[90,2] + -14.367;
   1:  PR[91,3] = PR[90,3] + 123.000;
   1:L PR[91] R[100]mm/sec CNT100;
   1:  PR[91,1] = PR[90,1] + 74.338;
   1:  PR[91,2] = PR[90,2] + -11.613;
   1:  PR[91,3] = PR[90,3] + 123.016;
   1:L PR[91] R[100]mm/sec CNT100;
   1:  PR[91,1] = PR[90,1] + 75.503;
   1:  PR[91,2] = PR[90,2] + -9.006;
   1:  PR[91,3] = PR[90,3] + 123.033;
   1:L PR[91] R[100]mm/sec CNT100;
   1:  PR[91,1] = PR[90,1] + 76.165;
   1:  PR[91,2] = PR[90,2] + -6.343;
   1:  PR[91,3] = PR[90,3] + 123.048;
   1:L PR[91] R[100]mm/sec CNT100;
   1:  PR[91,1] = PR[90,1] + 76.401;
   1:  PR[91,2] = PR[90,2] + -3.434;
   1:  PR[91,3] = PR[90,3] + 123.063;
   1:L PR[91] R[100]mm/sec CNT100;
   1:  PR[91,1] = PR[90,1] + 76.793;
   1:  PR[91,2] = PR[90,2] + -0.670;
   1:  PR[91,3] = PR[90,3] + 123.079;
   1:L PR[91] R[100]mm/sec CNT100;
   1:  PR[91,1] = PR[90,1] + 76.568;
   1:  PR[91,2] = PR[90,2] + 2.084;
   1:  PR[91,3] = PR[90,3] + 123.094;
   1:L PR[91] R[100]mm/sec CNT100;
   1:  PR[91,1] = PR[90,1] + 76.179;
   1:  PR[91,2] = PR[90,2] + 4.827;
   1:  PR[91,3] = PR[90,3] + 123.110;
   1:L PR[91] R[100]mm/sec CNT100;
   1:  PR[91,1] = PR[90,1] + 75.498;
   1:  PR[91,2] = PR[90,2] + 7.566;
   1:  PR[91,3] = PR[90,3] + 123.125;
   1:L PR[91] R[100]mm/sec CNT100;
   1:  PR[91,1] = PR[90,1] + 74.298;
   1:  PR[91,2] = PR[90,2] + 10.396;
   1:  PR[91,3] = PR[90,3] + 123.140;
   1:L PR[91] R[100]mm/sec CNT100;
   1:  PR[91,1] = PR[90,1] + 73.183;
   1:  PR[91,2] = PR[90,2] + 12.891;
   1:  PR[91,3] = PR[90,3] + 123.157;
   1:L PR[91] R[100]mm/sec CNT100;
   1:  PR[91,1] = PR[90,1] + 71.562;
   1:  PR[91,2] = PR[90,2] + 15.508;
   1:  PR[91,3] = PR[90,3] + 123.172;
   1:L PR[91] R[100]mm/sec CNT100;
   1:  PR[91,1] = PR[90,1] + 67.647;
   1:  PR[91,2] = PR[90,2] + 20.200;
   1:  PR[91,3] = PR[90,3] + 123.189;
   1:L PR[91] R[100]mm/sec CNT100;
   1:  PR[91,1] = PR[90,1] + 64.977;
   1:  PR[91,2] = PR[90,2] + 22.596;
   1:  PR[91,3] = PR[90,3] + 123.222;
   1:L PR[91] R[100]mm/sec CNT100;
   1:  PR[91,1] = PR[90,1] + 61.410;
   1:  PR[91,2] = PR[90,2] + 25.054;
   1:  PR[91,3] = PR[90,3] + 123.242;
   1:L PR[91] R[100]mm/sec CNT100;
   1:  PR[91,1] = PR[90,1] + 59.811;
   1:  PR[91,2] = PR[90,2] + 26.191;
   1:  PR[91,3] = PR[90,3] + 123.265;
   1:L PR[91] R[100]mm/sec CNT100;
   1:  PR[91,1] = PR[90,1] + 55.943;
   1:  PR[91,2] = PR[90,2] + 28.169;
   1:  PR[91,3] = PR[90,3] + 123.276;
   1:L PR[91] R[100]mm/sec CNT100;
   1:  PR[91,1] = PR[90,1] + 50.340;
   1:  PR[91,2] = PR[90,2] + 30.270;
   1:  PR[91,3] = PR[90,3] + 123.300;
   1:L PR[91] R[100]mm/sec CNT100;
   1:  PR[91,1] = PR[90,1] + 45.668;
   1:  PR[91,2] = PR[90,2] + 31.392;
   1:  PR[91,3] = PR[90,3] + 123.333;
   1:L PR[91] R[100]mm/sec CNT100;
   1:  PR[91,1] = PR[90,1] + 44.693;
   1:  PR[91,2] = PR[90,2] + 31.554;
   1:  PR[91,3] = PR[90,3] + 123.359;
   1:L PR[91] R[100]mm/sec CNT100;
   1:  PR[91,1] = PR[90,1] + 41.008;
   1:  PR[91,2] = PR[90,2] + 31.998;
   1:  PR[91,3] = PR[90,3] + 123.364;
   1:L PR[91] R[100]mm/sec CNT100;
   1:  PR[91,1] = PR[90,1] + 36.239;
   1:  PR[91,2] = PR[90,2] + 32.080;
   1:  PR[91,3] = PR[90,3] + 123.385;
   1:L PR[91] R[100]mm/sec CNT100;
   1:  PR[91,1] = PR[90,1] + 35.305;
   1:  PR[91,3] = PR[90,3] + 123.411;
   1:L PR[91] R[100]mm/sec CNT100;
   1:  PR[91,1] = PR[90,1] + 29.151;
   1:  PR[91,2] = PR[90,2] + 31.385;
   1:  PR[91,3] = PR[90,3] + 123.416;
   1:L PR[91] R[100]mm/sec CNT100;
   1:  PR[91,1] = PR[90,1] + 22.912;
   1:  PR[91,2] = PR[90,2] + 29.848;
   1:  PR[91,3] = PR[90,3] + 123.450;
   1:L PR[91] R[100]mm/sec CNT100;
   1:  PR[91,1] = PR[90,1] + 19.044;
   1:  PR[91,2] = PR[90,2] + 28.476;
   1:  PR[91,3] = PR[90,3] + 123.485;
   1:L PR[91] R[100]mm/sec CNT100;
   1:  PR[91,1] = PR[90,1] + 17.038;
   1:  PR[91,2] = PR[90,2] + 27.676;
   1:  PR[91,3] = PR[90,3] + 123.507;
   1:L PR[91] R[100]mm/sec CNT100;
   1:  PR[91,1] = PR[90,1] + 14.473;
   1:  PR[91,2] = PR[90,2] + 26.297;
   1:  PR[91,3] = PR[90,3] + 123.519;
   1:L PR[91] R[100]mm/sec CNT100;
   1:  PR[91,1] = PR[90,1] + 10.346;
   1:  PR[91,2] = PR[90,2] + 24.294;
   1:  PR[91,3] = PR[90,3] + 123.535;
   1:L PR[91] R[100]mm/sec CNT100;
   1:  PR[91,1] = PR[90,1] + 4.065;
   1:  PR[91,2] = PR[90,2] + 19.939;
   1:  PR[91,3] = PR[90,3] + 123.560;
   1:L PR[91] R[100]mm/sec CNT100;
   1:  PR[91,1] = PR[90,1] + 3.463;
   1:  PR[91,2] = PR[90,2] + 19.341;
   1:  PR[91,3] = PR[90,3] + 123.602;
   1:L PR[91] R[100]mm/sec CNT100;
   1:  PR[91,1] = PR[90,1] + -1.307;
   1:  PR[91,2] = PR[90,2] + 15.578;
   1:  PR[91,3] = PR[90,3] + 123.606;
   1:L PR[91] R[100]mm/sec CNT100;
   1:  PR[91,1] = PR[90,1] + -4.010;
   1:  PR[91,2] = PR[90,2] + 12.736;
   1:  PR[91,3] = PR[90,3] + 123.640;
   1:L PR[91] R[100]mm/sec CNT100;
   1:  PR[91,1] = PR[90,1] + -4.723;
   1:  PR[91,2] = PR[90,2] + 11.898;
   1:  PR[91,3] = PR[90,3] + 123.661;
   1:L PR[91] R[100]mm/sec CNT100;
   1:  PR[91,1] = PR[90,1] + -5.827;
   1:  PR[91,2] = PR[90,2] + 10.196;
   1:  PR[91,3] = PR[90,3] + 123.667;
   1:L PR[91] R[100]mm/sec CNT100;
   1:  PR[91,1] = PR[90,1] + -7.725;
   1:  PR[91,2] = PR[90,2] + 7.778;
   1:  PR[91,3] = PR[90,3] + 123.678;
   1:L PR[91] R[100]mm/sec CNT100;
   1:  PR[91] = PR[90];
   1:  PR[91,1] = PR[90,1] + -6.258;
   1:  PR[91,2] = PR[90,2] + 6.351;
   1:  PR[91,3] = PR[90,3] + 124.995;
   1:L PR[91] R[100]mm/sec CNT100;
   1:  PR[91,1] = PR[90,1] + -7.549;
   1:  PR[91,2] = PR[90,2] + 3.531;
   1:  PR[91,3] = PR[90,3] + 123.704;
   1:L PR[91] R[100]mm/sec CNT100;
   1:  PR[91,1] = PR[90,1] + -8.194;
   1:  PR[91,2] = PR[90,2] + -0.729;
   1:  PR[91,3] = PR[90,3] + 123.721;
   1:L PR[91] R[100]mm/sec CNT100;
   1:  PR[91,1] = PR[90,1] + -7.549;
   1:  PR[91,2] = PR[90,2] + -4.990;
   1:  PR[91,3] = PR[90,3] + 123.745;
   1:L PR[91] R[100]mm/sec CNT100;
   1:  PR[91,1] = PR[90,1] + -6.258;
   1:  PR[91,2] = PR[90,2] + -7.810;
   1:  PR[91,3] = PR[90,3] + 123.768;
   1:L PR[91] R[100]mm/sec CNT100;
   1:  PR[91,1] = PR[90,1] + -5.693;
   1:  PR[91,2] = PR[90,2] + -9.296;
   1:  PR[91,3] = PR[90,3] + 123.785;
   1:L PR[91] R[100]mm/sec CNT100;
   1:  PR[91,1] = PR[90,1] + -5.567;
   1:  PR[91,2] = PR[90,2] + -9.555;
   1:  PR[91,3] = PR[90,3] + 123.794;
   1:L PR[91] R[100]mm/sec CNT100;
   1:  PR[91,1] = PR[90,1] + -3.418;
   1:  PR[91,2] = PR[90,2] + -12.869;
   1:  PR[91,3] = PR[90,3] + 123.796;
   1:L PR[91] R[100]mm/sec CNT100;
   1:  PR[91,1] = PR[90,1] + -1.259;
   1:  PR[91,2] = PR[90,2] + -15.407;
   1:  PR[91,3] = PR[90,3] + 123.817;
   1:L PR[91] R[100]mm/sec CNT100;
   1:  PR[91,1] = PR[90,1] + 0.096;
   1:  PR[91,2] = PR[90,2] + -16.832;
   1:  PR[91,3] = PR[90,3] + 123.836;
   1:L PR[91] R[100]mm/sec CNT100;
   1:  PR[91,1] = PR[90,1] + 2.591;
   1:  PR[91,2] = PR[90,2] + -18.800;
   1:  PR[91,3] = PR[90,3] + 123.847;
   1:L PR[91] R[100]mm/sec CNT100;
   1:  PR[91,1] = PR[90,1] + 5.357;
   1:  PR[91,2] = PR[90,2] + -21.547;
   1:  PR[91,3] = PR[90,3] + 123.864;
   1:L PR[91] R[100]mm/sec CNT100;
   1:  PR[91,1] = PR[90,1] + 11.682;
   1:  PR[91,2] = PR[90,2] + -25.925;
   1:  PR[91,3] = PR[90,3] + 123.886;
   1:L PR[91] R[100]mm/sec CNT100;
   1:  PR[91,1] = PR[90,1] + 13.334;
   1:  PR[91,2] = PR[90,2] + -26.727;
   1:  PR[91,3] = PR[90,3] + 123.928;
   1:L PR[91] R[100]mm/sec CNT100;
   1:  PR[91,1] = PR[90,1] + 17.724;
   1:  PR[91,2] = PR[90,2] + -29.088;
   1:  PR[91,3] = PR[90,3] + 123.938;
   1:L PR[91] R[100]mm/sec CNT100;
   1:  PR[91,1] = PR[90,1] + 21.225;
   1:  PR[91,2] = PR[90,2] + -30.485;
   1:  PR[91,3] = PR[90,3] + 123.965;
   1:L PR[91] R[100]mm/sec CNT100;
   1:  PR[91,1] = PR[90,1] + 23.569;
   1:  PR[91,2] = PR[90,2] + -31.317;
   1:  PR[91,3] = PR[90,3] + 123.986;
   1:L PR[91] R[100]mm/sec CNT100;
   1:  PR[91,1] = PR[90,1] + 29.339;
   1:  PR[91,2] = PR[90,2] + -32.739;
